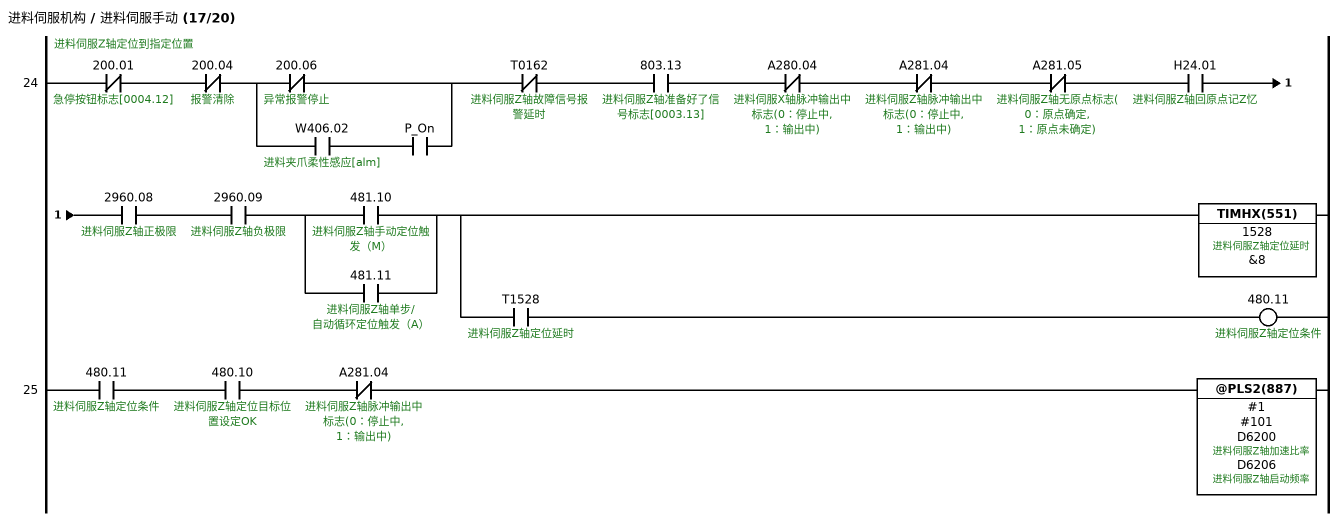
; [picture p96: 进料伺服机构 / 进料伺服手动, rungs 24-25]
; rung 24: 进料伺服Z轴定位到指定位置
LDNOT 200.01  ; 急停按钮标志[0004.12]
ANDNOT 200.04  ; 报警清除
LDNOT 200.06  ; 异常报警停止
LD W406.02  ; 进料夹爪柔性感应[alm]
AND P_On
ORLD
ANDLD
ANDNOT T0162  ; 进料伺服Z轴故障信号报警延时
AND 803.13  ; 进料伺服Z轴准备好了信号标志[0003.13]
ANDNOT A280.04  ; 进料伺服X轴脉冲输出中标志(0：停止中,1：输出中)
ANDNOT A281.04  ; 进料伺服Z轴脉冲输出中标志(0：停止中,1：输出中)
ANDNOT A281.05  ; 进料伺服Z轴无原点标志(0：原点确定,1：原点未确定)
AND H24.01  ; 进料伺服Z轴回原点记Z忆
AND 2960.08  ; 进料伺服Z轴正极限
AND 2960.09  ; 进料伺服Z轴负极限
LD 481.10  ; 进料伺服Z轴手动定位触发（M）
OR 481.11  ; 进料伺服Z轴单步/自动循环定位触发（A）
ANDLD
TIMHX(551) 1528 &8  ; 进料伺服Z轴定位延时
AND T1528  ; 进料伺服Z轴定位延时
OUT 480.11  ; 进料伺服Z轴定位条件
; rung 25
LD 480.11  ; 进料伺服Z轴定位条件
AND 480.10  ; 进料伺服Z轴定位目标位置设定OK
ANDNOT A281.04  ; 进料伺服Z轴脉冲输出中标志(0：停止中,1：输出中)
@PLS2(887) #1 #101 D6200 D6206  ; 进料伺服Z轴加速比率, 进料伺服Z轴启动频率

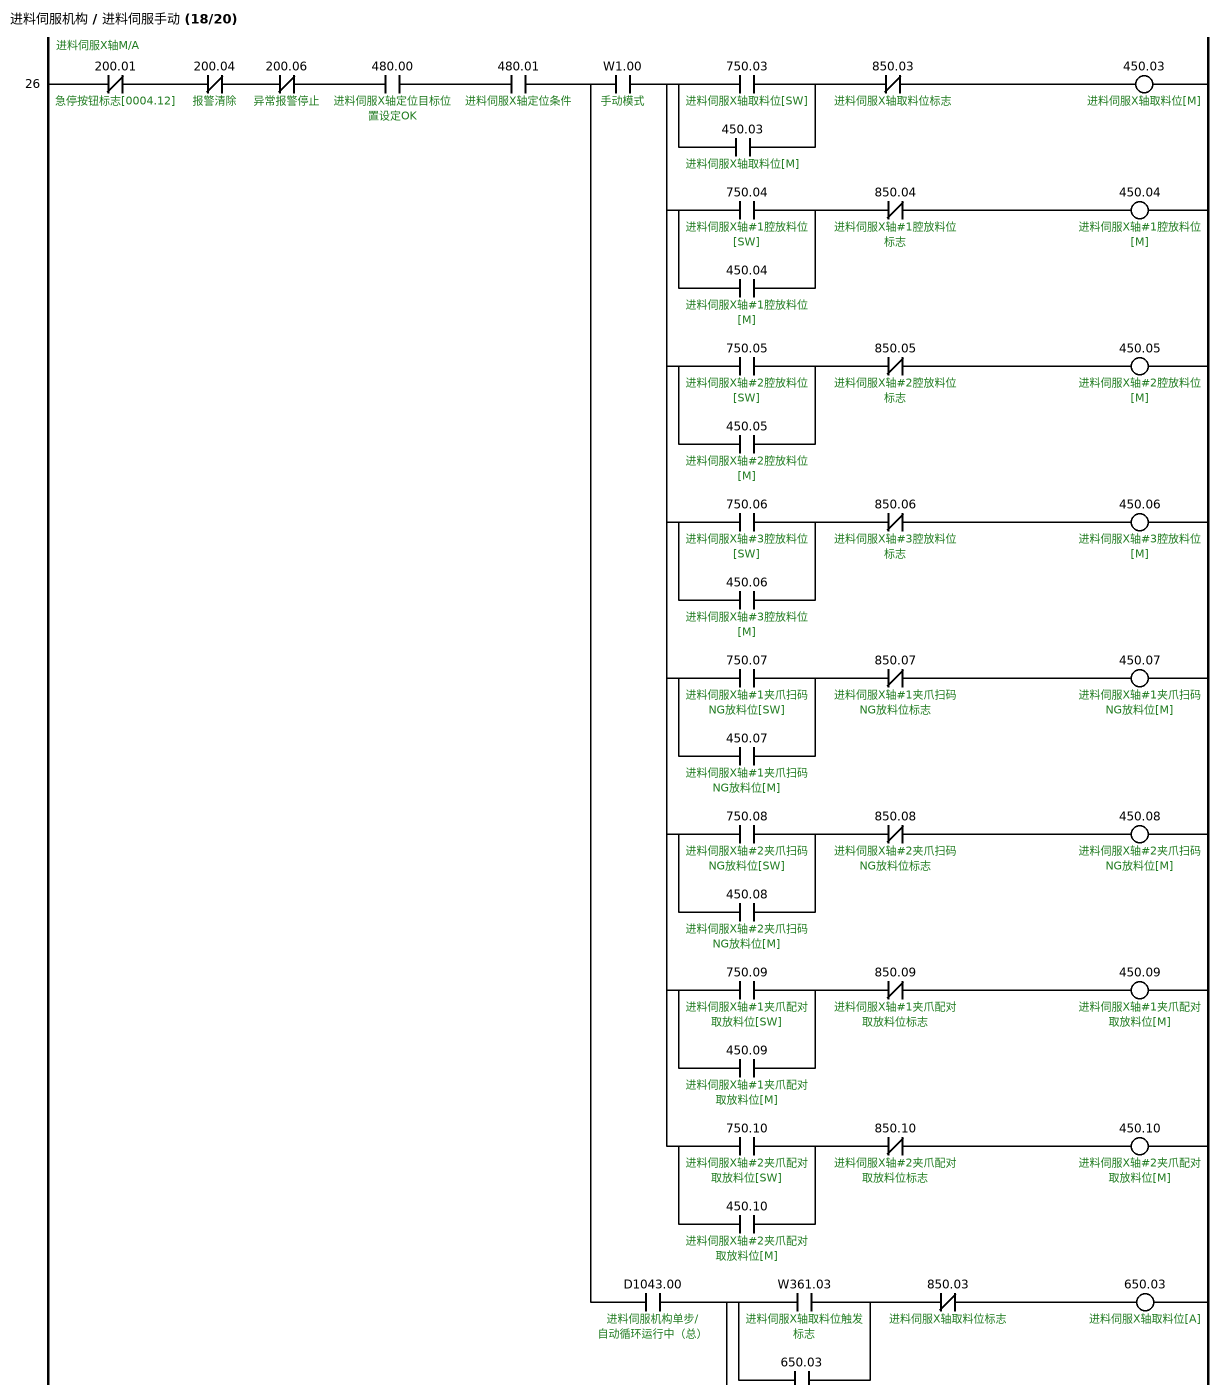

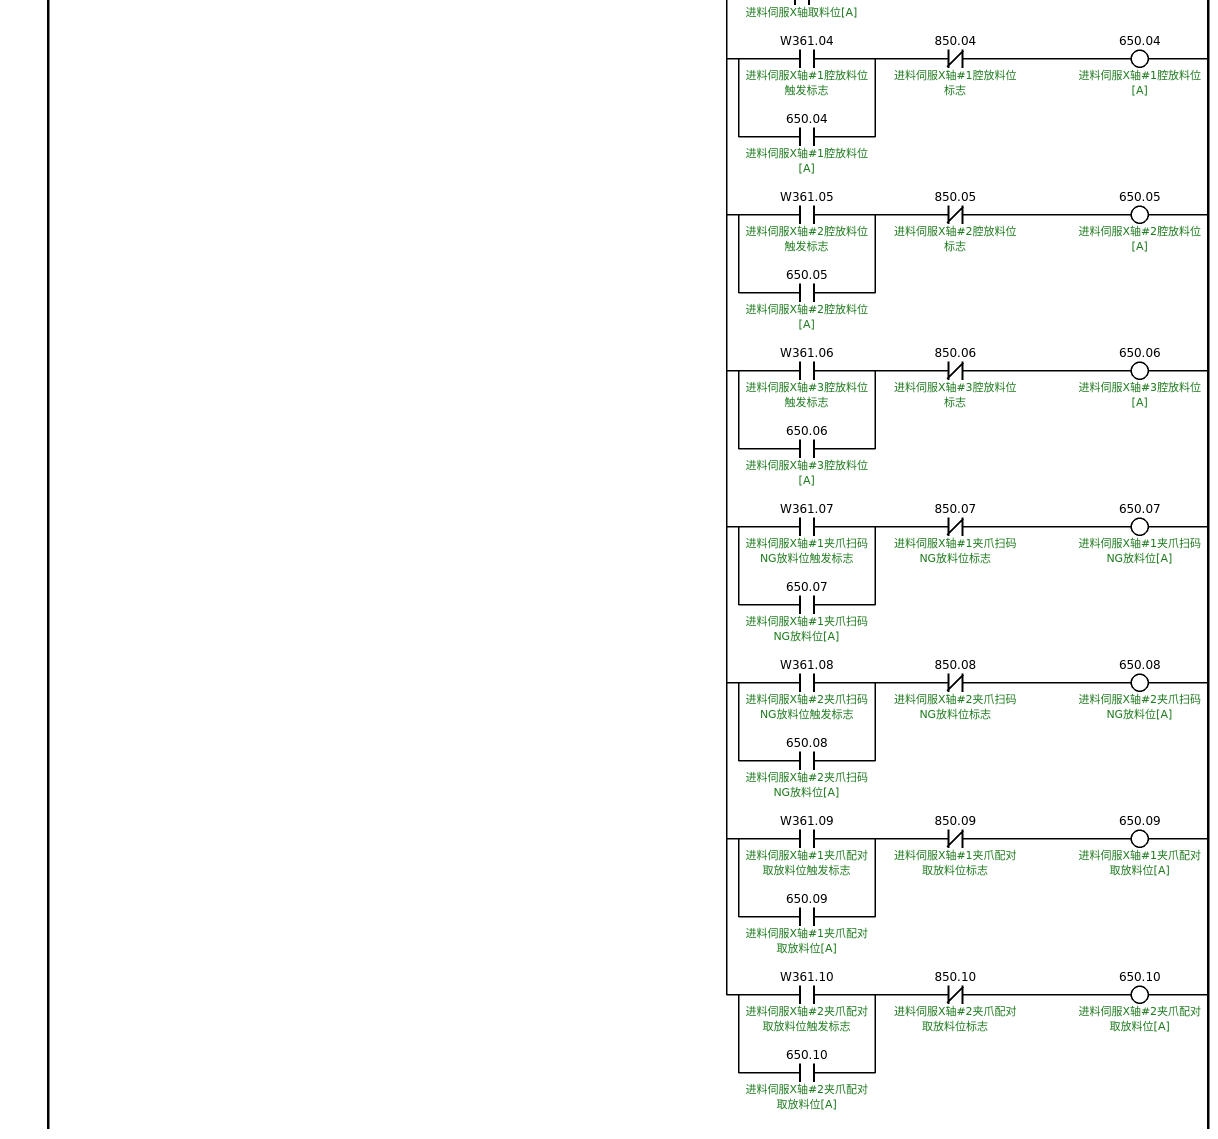
; rung 26: 进料伺服X轴M/A
LDNOT 200.01  ; 急停按钮标志[0004.12]
ANDNOT 200.04  ; 报警清除
ANDNOT 200.06  ; 异常报警停止
AND 480.00  ; 进料伺服X轴定位目标位置设定OK
AND 480.01  ; 进料伺服X轴定位条件
OUT TR0
AND W1.00  ; 手动模式
OUT TR1
LD 750.03  ; 进料伺服X轴取料位[SW]
OR 450.03  ; 进料伺服X轴取料位[M]
ANDLD
ANDNOT 850.03  ; 进料伺服X轴取料位标志
OUT 450.03  ; 进料伺服X轴取料位[M]
LD TR1
LD 750.04  ; 进料伺服X轴#1腔放料位[SW]
OR 450.04  ; 进料伺服X轴#1腔放料位[M]
ANDLD
ANDNOT 850.04  ; 进料伺服X轴#1腔放料位标志
OUT 450.04  ; 进料伺服X轴#1腔放料位[M]
LD TR1
LD 750.05  ; 进料伺服X轴#2腔放料位[SW]
OR 450.05  ; 进料伺服X轴#2腔放料位[M]
ANDLD
ANDNOT 850.05  ; 进料伺服X轴#2腔放料位标志
OUT 450.05  ; 进料伺服X轴#2腔放料位[M]
LD TR1
LD 750.06  ; 进料伺服X轴#3腔放料位[SW]
OR 450.06  ; 进料伺服X轴#3腔放料位[M]
ANDLD
ANDNOT 850.06  ; 进料伺服X轴#3腔放料位标志
OUT 450.06  ; 进料伺服X轴#3腔放料位[M]
LD TR1
LD 750.07  ; 进料伺服X轴#1夹爪扫码NG放料位[SW]
OR 450.07  ; 进料伺服X轴#1夹爪扫码NG放料位[M]
ANDLD
ANDNOT 850.07  ; 进料伺服X轴#1夹爪扫码NG放料位标志
OUT 450.07  ; 进料伺服X轴#1夹爪扫码NG放料位[M]
LD TR1
LD 750.08  ; 进料伺服X轴#2夹爪扫码NG放料位[SW]
OR 450.08  ; 进料伺服X轴#2夹爪扫码NG放料位[M]
ANDLD
ANDNOT 850.08  ; 进料伺服X轴#2夹爪扫码NG放料位标志
OUT 450.08  ; 进料伺服X轴#2夹爪扫码NG放料位[M]
LD TR1
LD 750.09  ; 进料伺服X轴#1夹爪配对取放料位[SW]
OR 450.09  ; 进料伺服X轴#1夹爪配对取放料位[M]
ANDLD
ANDNOT 850.09  ; 进料伺服X轴#1夹爪配对取放料位标志
OUT 450.09  ; 进料伺服X轴#1夹爪配对取放料位[M]
LD TR1
LD 750.10  ; 进料伺服X轴#2夹爪配对取放料位[SW]
OR 450.10  ; 进料伺服X轴#2夹爪配对取放料位[M]
ANDLD
ANDNOT 850.10  ; 进料伺服X轴#2夹爪配对取放料位标志
OUT 450.10  ; 进料伺服X轴#2夹爪配对取放料位[M]
LD TR0
AND D1043.00  ; 进料伺服机构单步/自动循环运行中（总）
OUT TR0
LD W361.03  ; 进料伺服X轴取料位触发标志
OR 650.03  ; 进料伺服X轴取料位[A]
ANDLD
ANDNOT 850.03  ; 进料伺服X轴取料位标志
OUT 650.03  ; 进料伺服X轴取料位[A]
LD TR0
LD W361.04  ; 进料伺服X轴#1腔放料位触发标志
OR 650.04  ; 进料伺服X轴#1腔放料位[A]
ANDLD
ANDNOT 850.04  ; 进料伺服X轴#1腔放料位标志
OUT 650.04  ; 进料伺服X轴#1腔放料位[A]
LD TR0
LD W361.05  ; 进料伺服X轴#2腔放料位触发标志
OR 650.05  ; 进料伺服X轴#2腔放料位[A]
ANDLD
ANDNOT 850.05  ; 进料伺服X轴#2腔放料位标志
OUT 650.05  ; 进料伺服X轴#2腔放料位[A]
LD TR0
LD W361.06  ; 进料伺服X轴#3腔放料位触发标志
OR 650.06  ; 进料伺服X轴#3腔放料位[A]
ANDLD
ANDNOT 850.06  ; 进料伺服X轴#3腔放料位标志
OUT 650.06  ; 进料伺服X轴#3腔放料位[A]
LD TR0
LD W361.07  ; 进料伺服X轴#1夹爪扫码NG放料位触发标志
OR 650.07  ; 进料伺服X轴#1夹爪扫码NG放料位[A]
ANDLD
ANDNOT 850.07  ; 进料伺服X轴#1夹爪扫码NG放料位标志
OUT 650.07  ; 进料伺服X轴#1夹爪扫码NG放料位[A]
LD TR0
LD W361.08  ; 进料伺服X轴#2夹爪扫码NG放料位触发标志
OR 650.08  ; 进料伺服X轴#2夹爪扫码NG放料位[A]
ANDLD
ANDNOT 850.08  ; 进料伺服X轴#2夹爪扫码NG放料位标志
OUT 650.08  ; 进料伺服X轴#2夹爪扫码NG放料位[A]
LD TR0
LD W361.09  ; 进料伺服X轴#1夹爪配对取放料位触发标志
OR 650.09  ; 进料伺服X轴#1夹爪配对取放料位[A]
ANDLD
ANDNOT 850.09  ; 进料伺服X轴#1夹爪配对取放料位标志
OUT 650.09  ; 进料伺服X轴#1夹爪配对取放料位[A]
LD TR0
LD W361.10  ; 进料伺服X轴#2夹爪配对取放料位触发标志
OR 650.10  ; 进料伺服X轴#2夹爪配对取放料位[A]
ANDLD
ANDNOT 850.10  ; 进料伺服X轴#2夹爪配对取放料位标志
OUT 650.10  ; 进料伺服X轴#2夹爪配对取放料位[A]

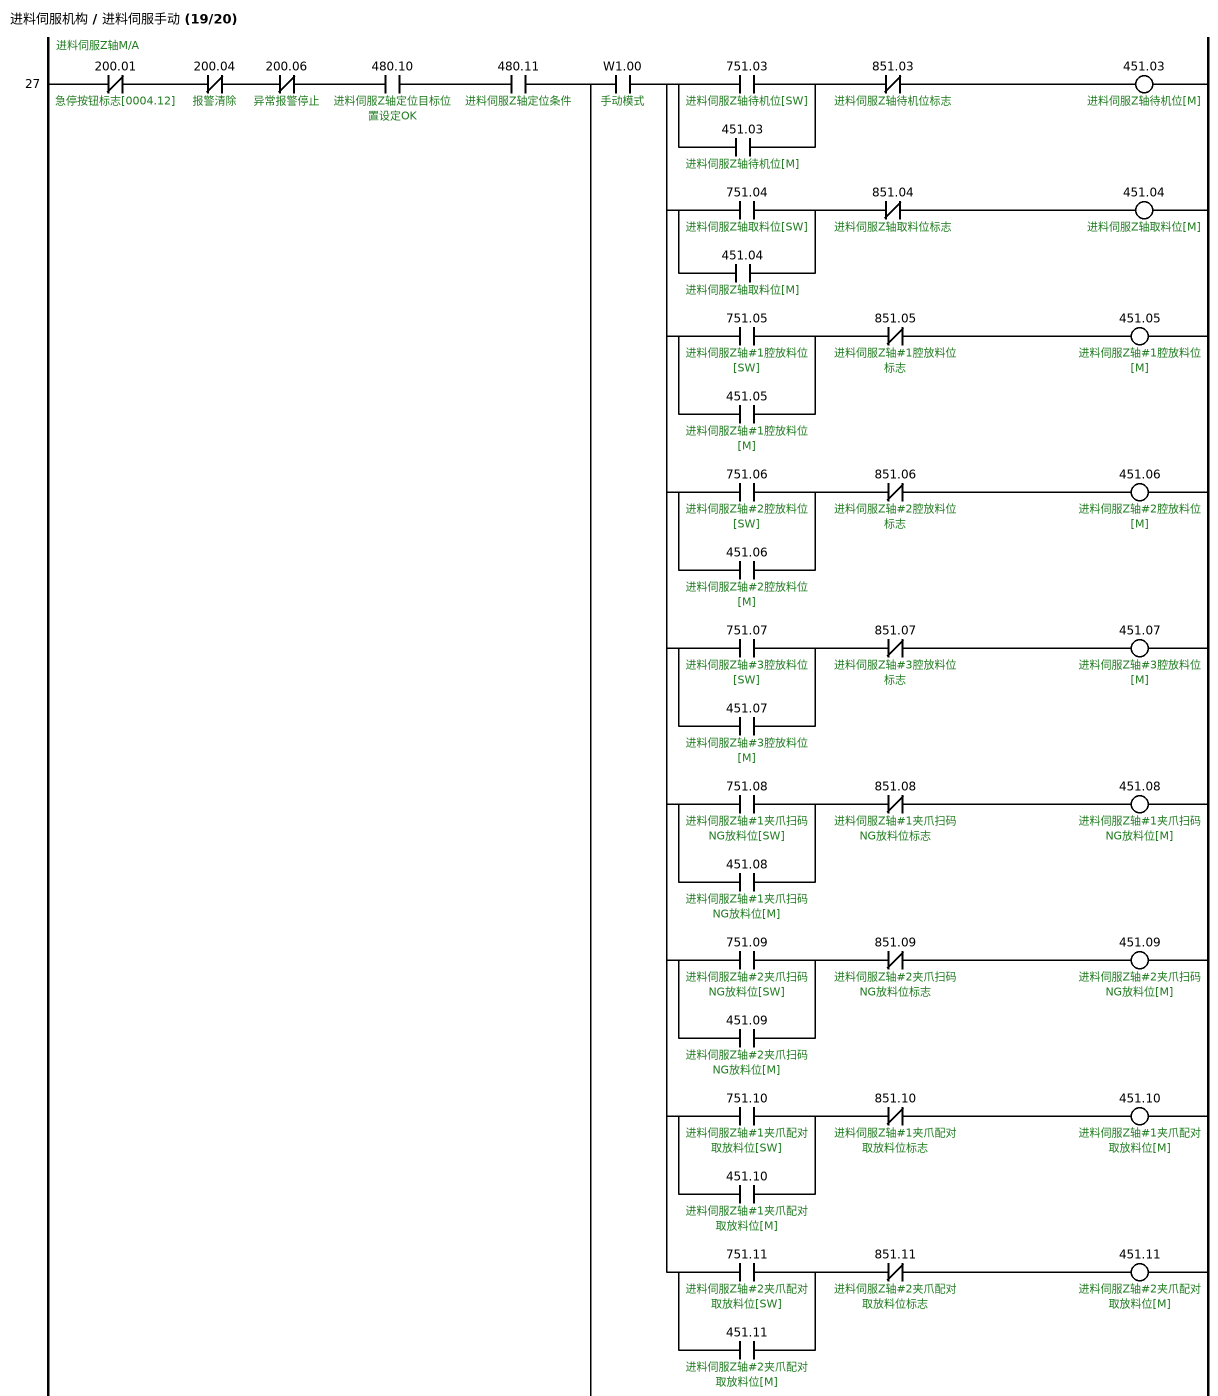

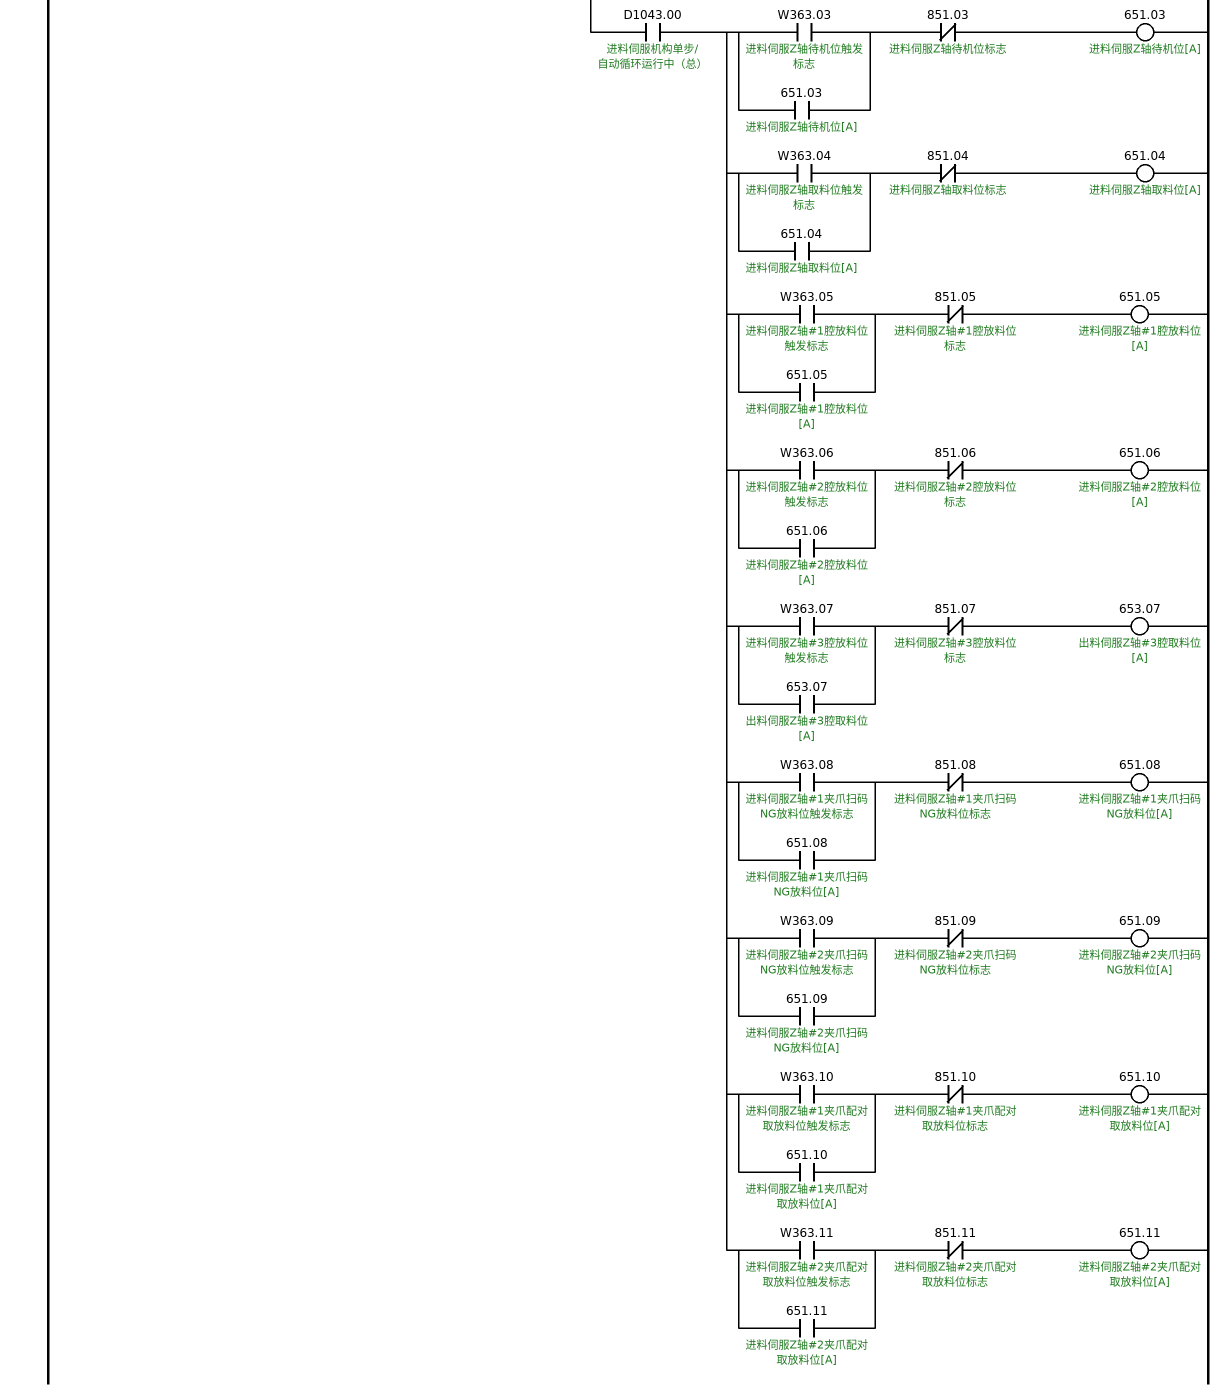
; rung 27: 进料伺服Z轴M/A
LDNOT 200.01  ; 急停按钮标志[0004.12]
ANDNOT 200.04  ; 报警清除
ANDNOT 200.06  ; 异常报警停止
AND 480.10  ; 进料伺服Z轴定位目标位置设定OK
AND 480.11  ; 进料伺服Z轴定位条件
OUT TR0
AND W1.00  ; 手动模式
OUT TR1
LD 751.03  ; 进料伺服Z轴待机位[SW]
OR 451.03  ; 进料伺服Z轴待机位[M]
ANDLD
ANDNOT 851.03  ; 进料伺服Z轴待机位标志
OUT 451.03  ; 进料伺服Z轴待机位[M]
LD TR1
LD 751.04  ; 进料伺服Z轴取料位[SW]
OR 451.04  ; 进料伺服Z轴取料位[M]
ANDLD
ANDNOT 851.04  ; 进料伺服Z轴取料位标志
OUT 451.04  ; 进料伺服Z轴取料位[M]
LD TR1
LD 751.05  ; 进料伺服Z轴#1腔放料位[SW]
OR 451.05  ; 进料伺服Z轴#1腔放料位[M]
ANDLD
ANDNOT 851.05  ; 进料伺服Z轴#1腔放料位标志
OUT 451.05  ; 进料伺服Z轴#1腔放料位[M]
LD TR1
LD 751.06  ; 进料伺服Z轴#2腔放料位[SW]
OR 451.06  ; 进料伺服Z轴#2腔放料位[M]
ANDLD
ANDNOT 851.06  ; 进料伺服Z轴#2腔放料位标志
OUT 451.06  ; 进料伺服Z轴#2腔放料位[M]
LD TR1
LD 751.07  ; 进料伺服Z轴#3腔放料位[SW]
OR 451.07  ; 进料伺服Z轴#3腔放料位[M]
ANDLD
ANDNOT 851.07  ; 进料伺服Z轴#3腔放料位标志
OUT 451.07  ; 进料伺服Z轴#3腔放料位[M]
LD TR1
LD 751.08  ; 进料伺服Z轴#1夹爪扫码NG放料位[SW]
OR 451.08  ; 进料伺服Z轴#1夹爪扫码NG放料位[M]
ANDLD
ANDNOT 851.08  ; 进料伺服Z轴#1夹爪扫码NG放料位标志
OUT 451.08  ; 进料伺服Z轴#1夹爪扫码NG放料位[M]
LD TR1
LD 751.09  ; 进料伺服Z轴#2夹爪扫码NG放料位[SW]
OR 451.09  ; 进料伺服Z轴#2夹爪扫码NG放料位[M]
ANDLD
ANDNOT 851.09  ; 进料伺服Z轴#2夹爪扫码NG放料位标志
OUT 451.09  ; 进料伺服Z轴#2夹爪扫码NG放料位[M]
LD TR1
LD 751.10  ; 进料伺服Z轴#1夹爪配对取放料位[SW]
OR 451.10  ; 进料伺服Z轴#1夹爪配对取放料位[M]
ANDLD
ANDNOT 851.10  ; 进料伺服Z轴#1夹爪配对取放料位标志
OUT 451.10  ; 进料伺服Z轴#1夹爪配对取放料位[M]
LD TR1
LD 751.11  ; 进料伺服Z轴#2夹爪配对取放料位[SW]
OR 451.11  ; 进料伺服Z轴#2夹爪配对取放料位[M]
ANDLD
ANDNOT 851.11  ; 进料伺服Z轴#2夹爪配对取放料位标志
OUT 451.11  ; 进料伺服Z轴#2夹爪配对取放料位[M]
LD TR0
AND D1043.00  ; 进料伺服机构单步/自动循环运行中（总）
OUT TR0
LD W363.03  ; 进料伺服Z轴待机位触发标志
OR 651.03  ; 进料伺服Z轴待机位[A]
ANDLD
ANDNOT 851.03  ; 进料伺服Z轴待机位标志
OUT 651.03  ; 进料伺服Z轴待机位[A]
LD TR0
LD W363.04  ; 进料伺服Z轴取料位触发标志
OR 651.04  ; 进料伺服Z轴取料位[A]
ANDLD
ANDNOT 851.04  ; 进料伺服Z轴取料位标志
OUT 651.04  ; 进料伺服Z轴取料位[A]
LD TR0
LD W363.05  ; 进料伺服Z轴#1腔放料位触发标志
OR 651.05  ; 进料伺服Z轴#1腔放料位[A]
ANDLD
ANDNOT 851.05  ; 进料伺服Z轴#1腔放料位标志
OUT 651.05  ; 进料伺服Z轴#1腔放料位[A]
LD TR0
LD W363.06  ; 进料伺服Z轴#2腔放料位触发标志
OR 651.06  ; 进料伺服Z轴#2腔放料位[A]
ANDLD
ANDNOT 851.06  ; 进料伺服Z轴#2腔放料位标志
OUT 651.06  ; 进料伺服Z轴#2腔放料位[A]
LD TR0
LD W363.07  ; 进料伺服Z轴#3腔放料位触发标志
OR 653.07  ; 出料伺服Z轴#3腔取料位[A]
ANDLD
ANDNOT 851.07  ; 进料伺服Z轴#3腔放料位标志
OUT 653.07  ; 出料伺服Z轴#3腔取料位[A]
LD TR0
LD W363.08  ; 进料伺服Z轴#1夹爪扫码NG放料位触发标志
OR 651.08  ; 进料伺服Z轴#1夹爪扫码NG放料位[A]
ANDLD
ANDNOT 851.08  ; 进料伺服Z轴#1夹爪扫码NG放料位标志
OUT 651.08  ; 进料伺服Z轴#1夹爪扫码NG放料位[A]
LD TR0
LD W363.09  ; 进料伺服Z轴#2夹爪扫码NG放料位触发标志
OR 651.09  ; 进料伺服Z轴#2夹爪扫码NG放料位[A]
ANDLD
ANDNOT 851.09  ; 进料伺服Z轴#2夹爪扫码NG放料位标志
OUT 651.09  ; 进料伺服Z轴#2夹爪扫码NG放料位[A]
LD TR0
LD W363.10  ; 进料伺服Z轴#1夹爪配对取放料位触发标志
OR 651.10  ; 进料伺服Z轴#1夹爪配对取放料位[A]
ANDLD
ANDNOT 851.10  ; 进料伺服Z轴#1夹爪配对取放料位标志
OUT 651.10  ; 进料伺服Z轴#1夹爪配对取放料位[A]
LD TR0
LD W363.11  ; 进料伺服Z轴#2夹爪配对取放料位触发标志
OR 651.11  ; 进料伺服Z轴#2夹爪配对取放料位[A]
ANDLD
ANDNOT 851.11  ; 进料伺服Z轴#2夹爪配对取放料位标志
OUT 651.11  ; 进料伺服Z轴#2夹爪配对取放料位[A]

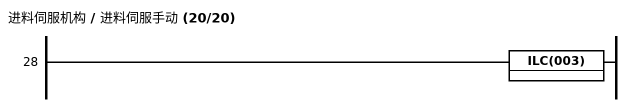
; rung 28
ILC(003)

### Section 进料伺服自动

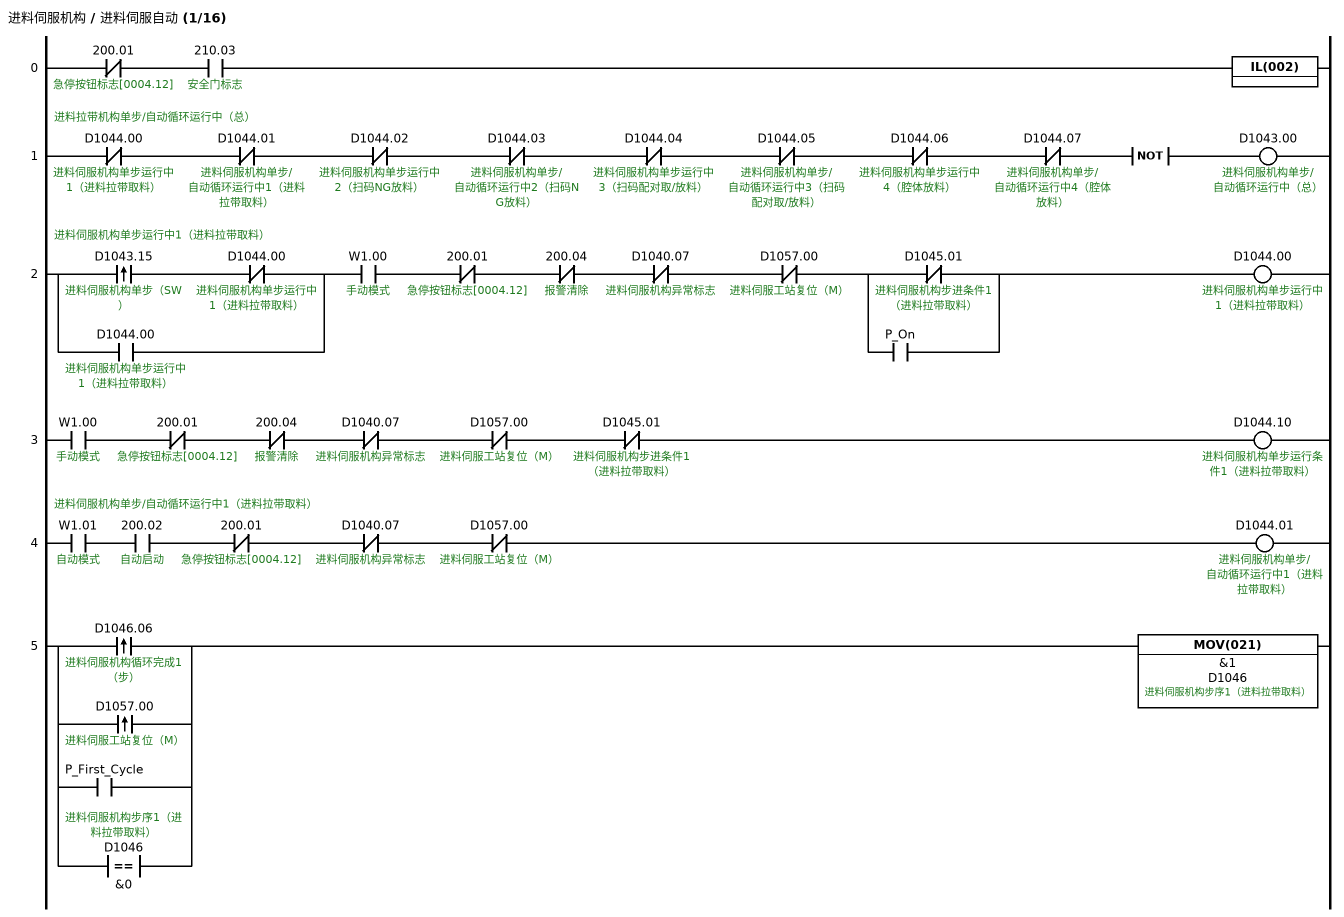
; rung 0
LDNOT 200.01  ; 急停按钮标志[0004.12]
AND 210.03  ; 安全门标志
IL(002)
; rung 1: 进料拉带机构单步/自动循环运行中（总）
LDNOT D1044.00  ; 进料伺服机构单步运行中1（进料拉带取料）
ANDNOT D1044.01  ; 进料伺服机构单步/自动循环运行中1（进料拉带取料）
ANDNOT D1044.02  ; 进料伺服机构单步运行中2（扫码NG放料）
ANDNOT D1044.03  ; 进料伺服机构单步/自动循环运行中2（扫码NG放料）
ANDNOT D1044.04  ; 进料伺服机构单步运行中3（扫码配对取/放料）
ANDNOT D1044.05  ; 进料伺服机构单步/自动循环运行中3（扫码配对取/放料）
ANDNOT D1044.06  ; 进料伺服机构单步运行中4（腔体放料）
ANDNOT D1044.07  ; 进料伺服机构单步/自动循环运行中4（腔体放料）
NOT(520)
OUT D1043.00  ; 进料伺服机构单步/自动循环运行中（总）
; rung 2: 进料伺服机构单步运行中1（进料拉带取料）
@LD D1043.15  ; 进料伺服机构单步（SW）
ANDNOT D1044.00  ; 进料伺服机构单步运行中1（进料拉带取料）
OR D1044.00  ; 进料伺服机构单步运行中1（进料拉带取料）
AND W1.00  ; 手动模式
ANDNOT 200.01  ; 急停按钮标志[0004.12]
ANDNOT 200.04  ; 报警清除
ANDNOT D1040.07  ; 进料伺服机构异常标志
ANDNOT D1057.00  ; 进料伺服工站复位（M）
LDNOT D1045.01  ; 进料伺服机构步进条件1（进料拉带取料）
OR P_On
ANDLD
OUT D1044.00  ; 进料伺服机构单步运行中1（进料拉带取料）
; rung 3
LD W1.00  ; 手动模式
ANDNOT 200.01  ; 急停按钮标志[0004.12]
ANDNOT 200.04  ; 报警清除
ANDNOT D1040.07  ; 进料伺服机构异常标志
ANDNOT D1057.00  ; 进料伺服工站复位（M）
ANDNOT D1045.01  ; 进料伺服机构步进条件1（进料拉带取料）
OUT D1044.10  ; 进料伺服机构单步运行条件1（进料拉带取料）
; rung 4: 进料伺服机构单步/自动循环运行中1（进料拉带取料）
LD W1.01  ; 自动模式
AND 200.02  ; 自动启动
ANDNOT 200.01  ; 急停按钮标志[0004.12]
ANDNOT D1040.07  ; 进料伺服机构异常标志
ANDNOT D1057.00  ; 进料伺服工站复位（M）
OUT D1044.01  ; 进料伺服机构单步/自动循环运行中1（进料拉带取料）
; rung 5
@LD D1046.06  ; 进料伺服机构循环完成1（步）
@OR D1057.00  ; 进料伺服工站复位（M）
OR P_First_Cycle
OR=(300) D1046 &0  ; 进料伺服机构步序1（进料拉带取料）
MOV(021) &1 D1046  ; 进料伺服机构步序1（进料拉带取料）

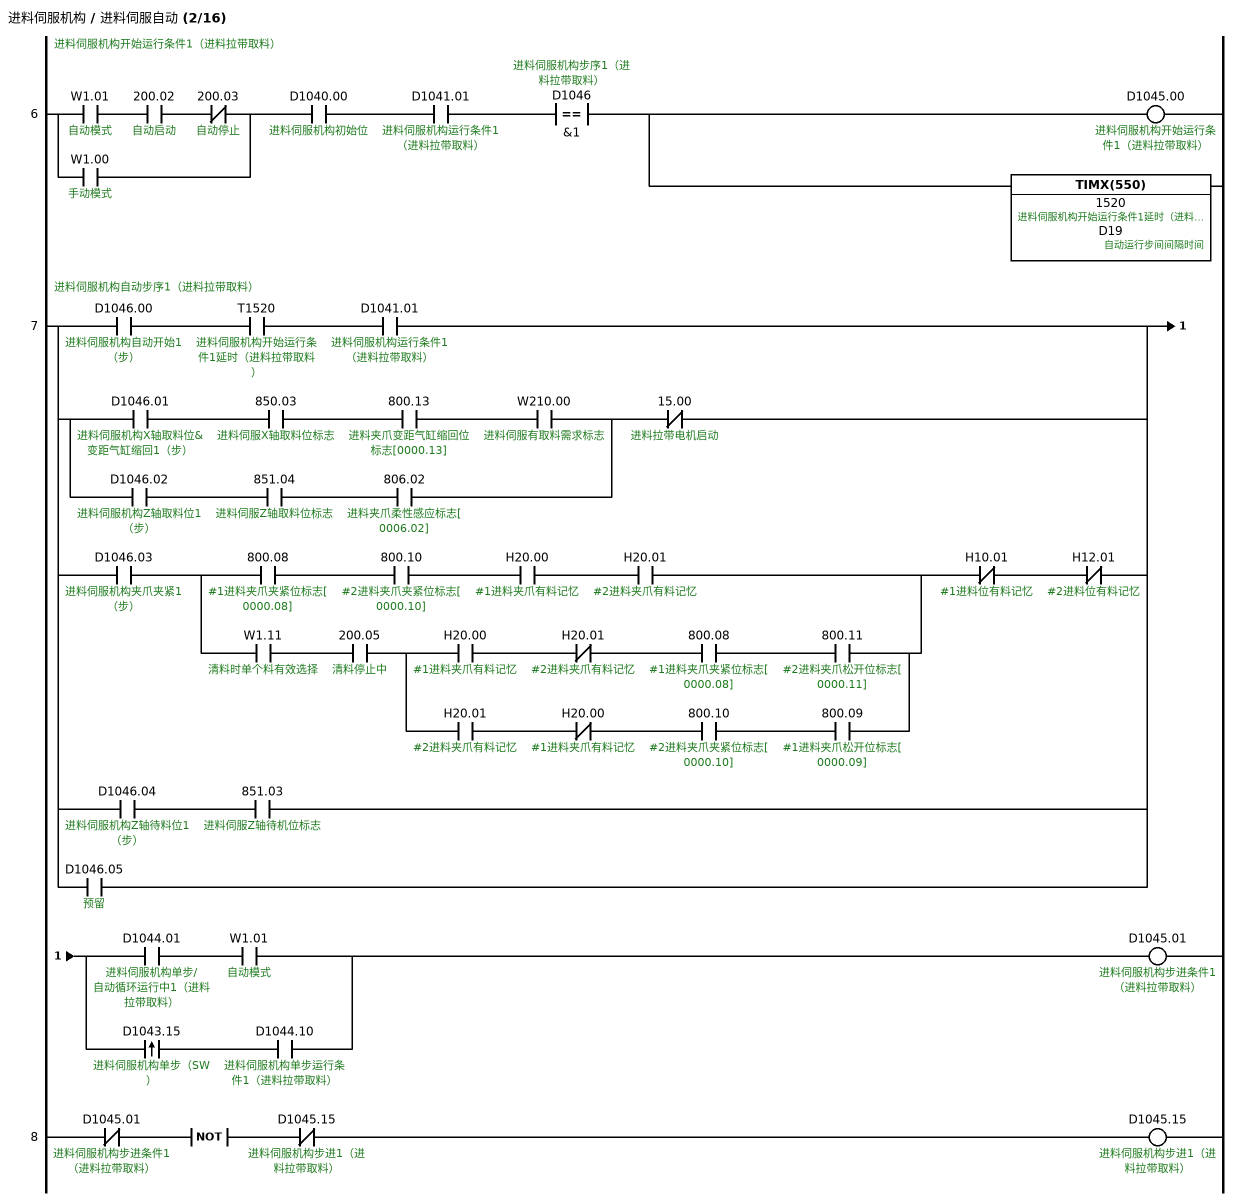
; rung 6: 进料伺服机构开始运行条件1（进料拉带取料）
LD W1.01  ; 自动模式
AND 200.02  ; 自动启动
ANDNOT 200.03  ; 自动停止
OR W1.00  ; 手动模式
AND D1040.00  ; 进料伺服机构初始位
AND D1041.01  ; 进料伺服机构运行条件1（进料拉带取料）
AND=(300) D1046 &1  ; 进料伺服机构步序1（进料拉带取料）
OUT D1045.00  ; 进料伺服机构开始运行条件1（进料拉带取料）
TIMX(550) 1520 D19  ; 自动运行步间间隔时间, 进料伺服机构开始运行条件1延时（进料拉带取料）
; rung 7: 进料伺服机构自动步序1（进料拉带取料）
LD D1046.00  ; 进料伺服机构自动开始1（步）
AND T1520  ; 进料伺服机构开始运行条件1延时（进料拉带取料）
AND D1041.01  ; 进料伺服机构运行条件1（进料拉带取料）
LD D1046.01  ; 进料伺服机构X轴取料位&变距气缸缩回1（步）
AND 850.03  ; 进料伺服X轴取料位标志
AND 800.13  ; 进料夹爪变距气缸缩回位标志[0000.13]
AND W210.00  ; 进料伺服有取料需求标志
LD D1046.02  ; 进料伺服机构Z轴取料位1（步）
AND 851.04  ; 进料伺服Z轴取料位标志
AND 806.02  ; 进料夹爪柔性感应标志[0006.02]
ORLD
ANDNOT 15.00  ; 进料拉带电机启动
ORLD
LD D1046.03  ; 进料伺服机构夹爪夹紧1（步）
LD 800.08  ; #1进料夹爪夹紧位标志[0000.08]
AND 800.10  ; #2进料夹爪夹紧位标志[0000.10]
AND H20.00  ; #1进料夹爪有料记忆
AND H20.01  ; #2进料夹爪有料记忆
LD W1.11  ; 清料时单个料有效选择
AND 200.05  ; 清料停止中
LD H20.00  ; #1进料夹爪有料记忆
ANDNOT H20.01  ; #2进料夹爪有料记忆
AND 800.08  ; #1进料夹爪夹紧位标志[0000.08]
AND 800.11  ; #2进料夹爪松开位标志[0000.11]
LD H20.01  ; #2进料夹爪有料记忆
ANDNOT H20.00  ; #1进料夹爪有料记忆
AND 800.10  ; #2进料夹爪夹紧位标志[0000.10]
AND 800.09  ; #1进料夹爪松开位标志[0000.09]
ORLD
ANDLD
ORLD
ANDLD
ANDNOT H10.01  ; #1进料位有料记忆
ANDNOT H12.01  ; #2进料位有料记忆
ORLD
LD D1046.04  ; 进料伺服机构Z轴待料位1（步）
AND 851.03  ; 进料伺服Z轴待机位标志
ORLD
OR D1046.05  ; 预留
LD D1044.01  ; 进料伺服机构单步/自动循环运行中1（进料拉带取料）
AND W1.01  ; 自动模式
@LD D1043.15  ; 进料伺服机构单步（SW）
AND D1044.10  ; 进料伺服机构单步运行条件1（进料拉带取料）
ORLD
ANDLD
OUT D1045.01  ; 进料伺服机构步进条件1（进料拉带取料）
; rung 8
LDNOT D1045.01  ; 进料伺服机构步进条件1（进料拉带取料）
NOT(520)
ANDNOT D1045.15  ; 进料伺服机构步进1（进料拉带取料）
OUT D1045.15  ; 进料伺服机构步进1（进料拉带取料）

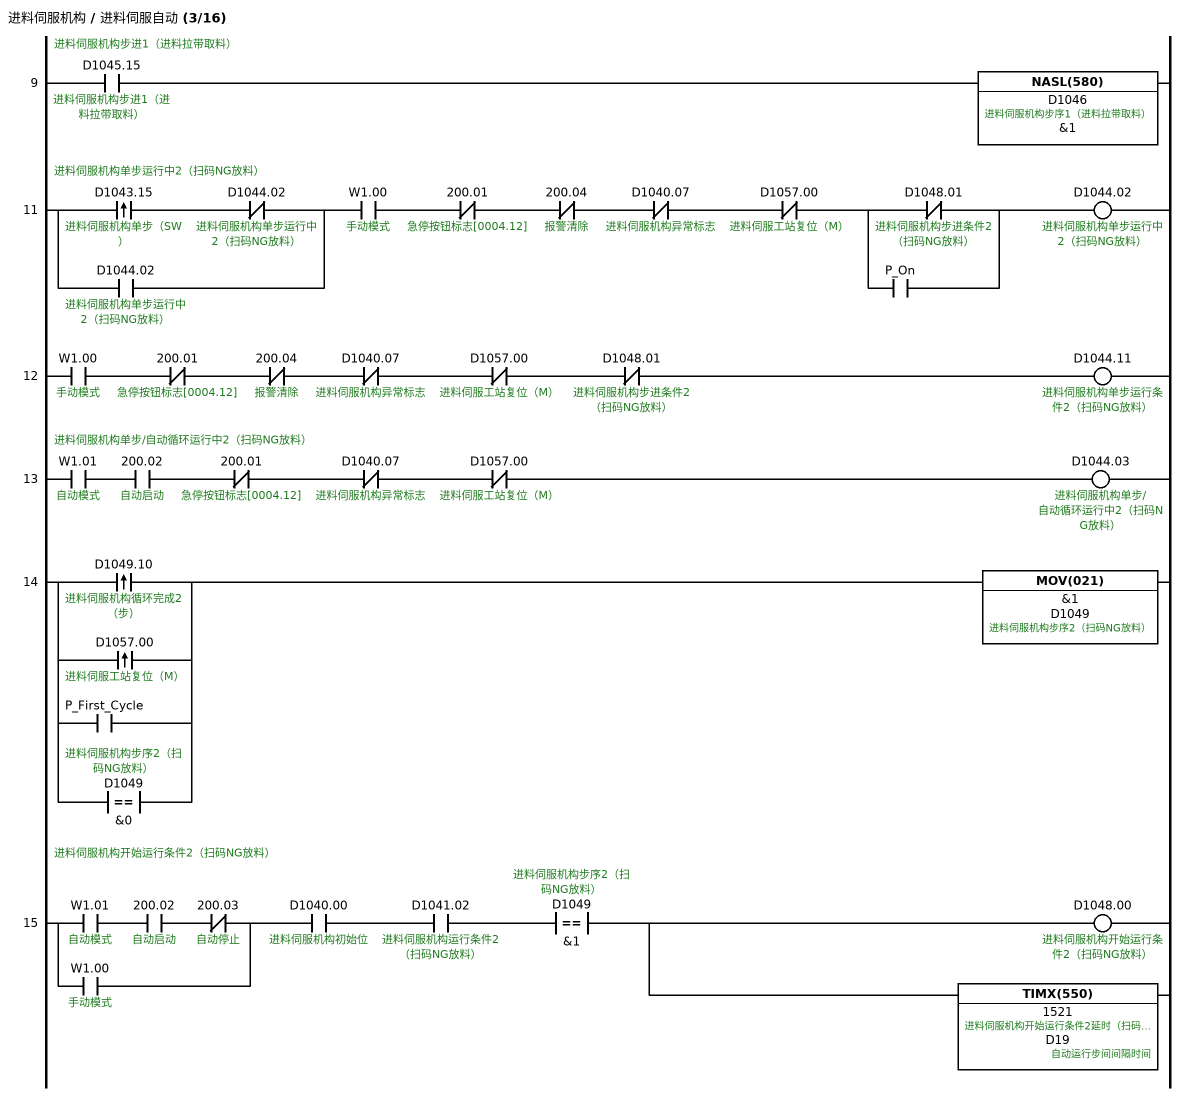
; rung 9: 进料伺服机构步进1（进料拉带取料）
LD D1045.15  ; 进料伺服机构步进1（进料拉带取料）
NASL(580) D1046 &1  ; 进料伺服机构步序1（进料拉带取料）
; rung 10: 进料伺服机构步序跳转程序1（进料拉带取料）
; rung 11: 进料伺服机构单步运行中2（扫码NG放料）
@LD D1043.15  ; 进料伺服机构单步（SW）
ANDNOT D1044.02  ; 进料伺服机构单步运行中2（扫码NG放料）
OR D1044.02  ; 进料伺服机构单步运行中2（扫码NG放料）
AND W1.00  ; 手动模式
ANDNOT 200.01  ; 急停按钮标志[0004.12]
ANDNOT 200.04  ; 报警清除
ANDNOT D1040.07  ; 进料伺服机构异常标志
ANDNOT D1057.00  ; 进料伺服工站复位（M）
LDNOT D1048.01  ; 进料伺服机构步进条件2（扫码NG放料）
OR P_On
ANDLD
OUT D1044.02  ; 进料伺服机构单步运行中2（扫码NG放料）
; rung 12
LD W1.00  ; 手动模式
ANDNOT 200.01  ; 急停按钮标志[0004.12]
ANDNOT 200.04  ; 报警清除
ANDNOT D1040.07  ; 进料伺服机构异常标志
ANDNOT D1057.00  ; 进料伺服工站复位（M）
ANDNOT D1048.01  ; 进料伺服机构步进条件2（扫码NG放料）
OUT D1044.11  ; 进料伺服机构单步运行条件2（扫码NG放料）
; rung 13: 进料伺服机构单步/自动循环运行中2（扫码NG放料）
LD W1.01  ; 自动模式
AND 200.02  ; 自动启动
ANDNOT 200.01  ; 急停按钮标志[0004.12]
ANDNOT D1040.07  ; 进料伺服机构异常标志
ANDNOT D1057.00  ; 进料伺服工站复位（M）
OUT D1044.03  ; 进料伺服机构单步/自动循环运行中2（扫码NG放料）
; rung 14
@LD D1049.10  ; 进料伺服机构循环完成2（步）
@OR D1057.00  ; 进料伺服工站复位（M）
OR P_First_Cycle
OR=(300) D1049 &0  ; 进料伺服机构步序2（扫码NG放料）
MOV(021) &1 D1049  ; 进料伺服机构步序2（扫码NG放料）
; rung 15: 进料伺服机构开始运行条件2（扫码NG放料）
LD W1.01  ; 自动模式
AND 200.02  ; 自动启动
ANDNOT 200.03  ; 自动停止
OR W1.00  ; 手动模式
AND D1040.00  ; 进料伺服机构初始位
AND D1041.02  ; 进料伺服机构运行条件2（扫码NG放料）
AND=(300) D1049 &1  ; 进料伺服机构步序2（扫码NG放料）
OUT D1048.00  ; 进料伺服机构开始运行条件2（扫码NG放料）
TIMX(550) 1521 D19  ; 自动运行步间间隔时间, 进料伺服机构开始运行条件2延时（扫码NG放料）

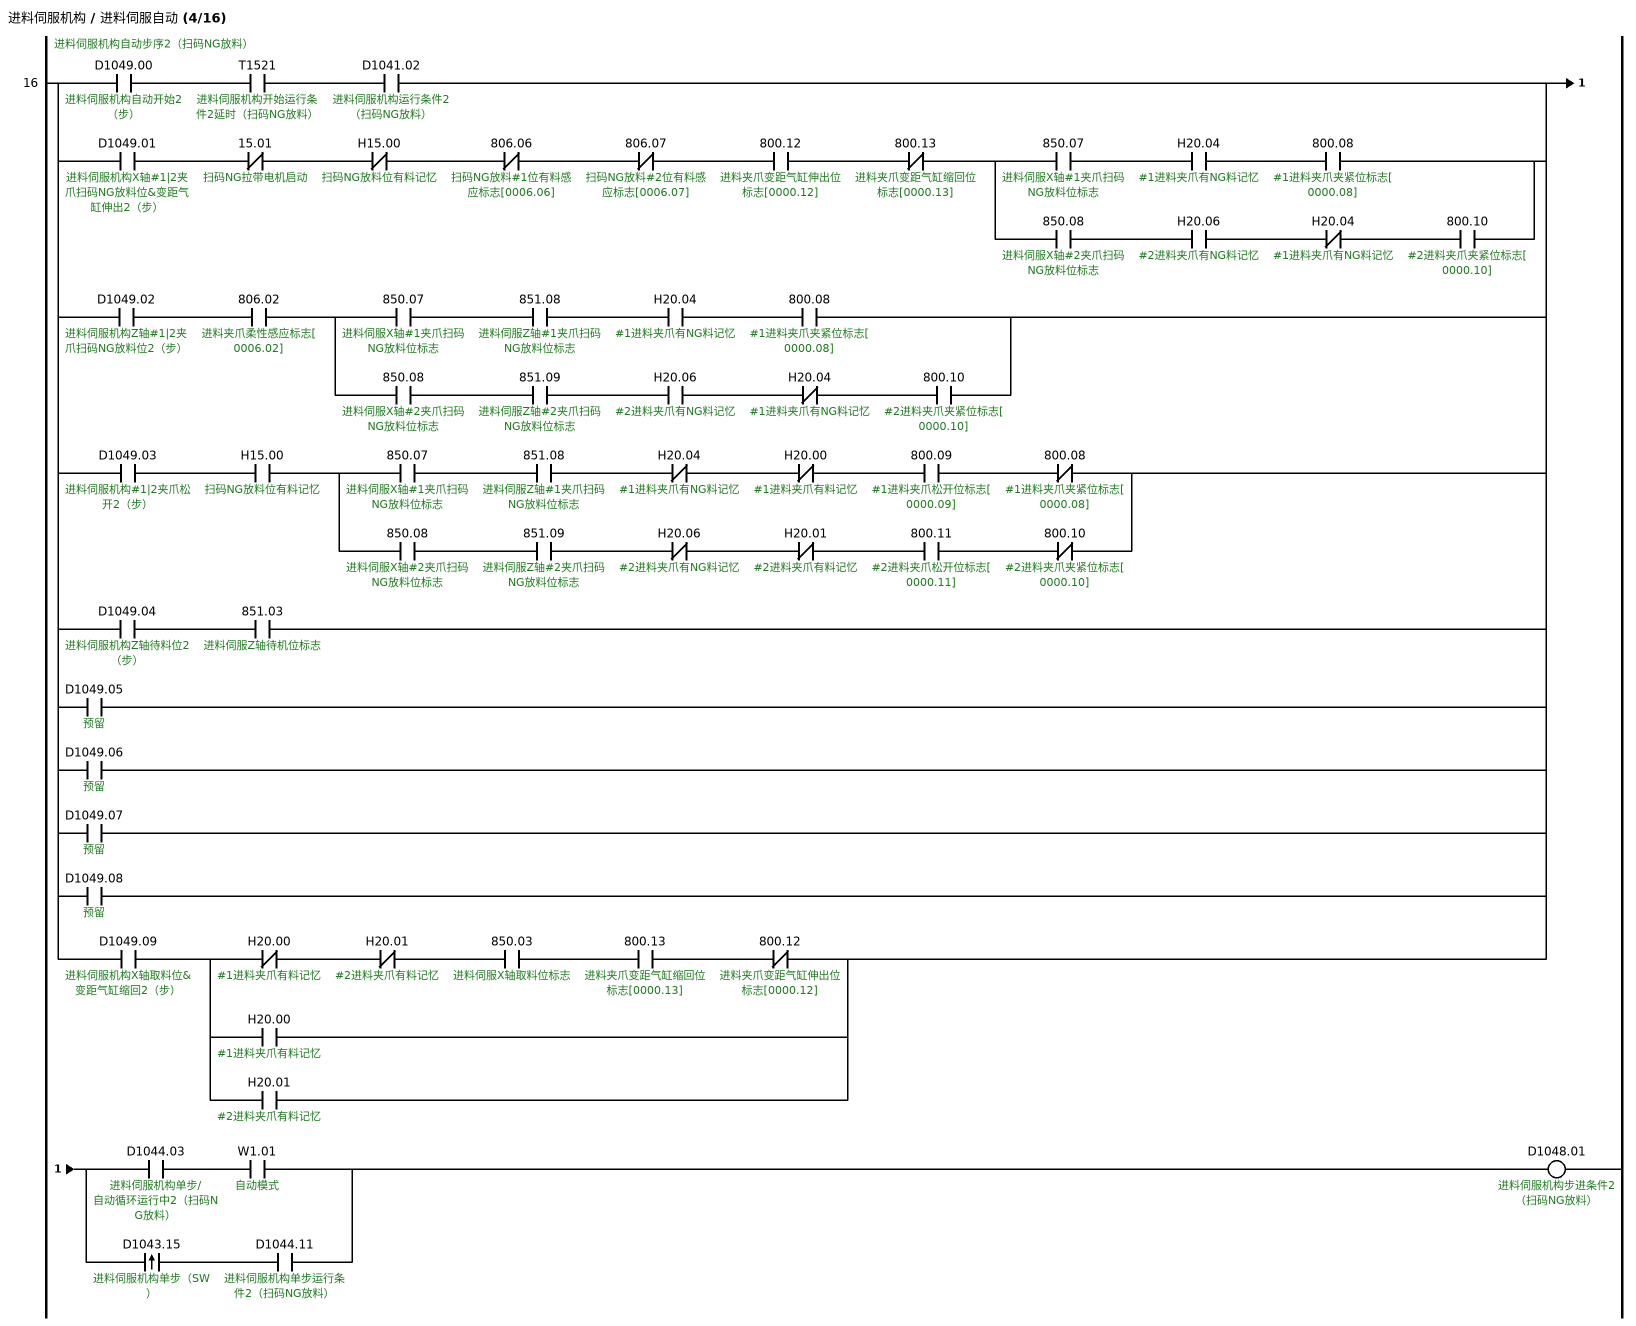
; rung 16: 进料伺服机构自动步序2（扫码NG放料）
LD D1049.00  ; 进料伺服机构自动开始2（步）
AND T1521  ; 进料伺服机构开始运行条件2延时（扫码NG放料）
AND D1041.02  ; 进料伺服机构运行条件2（扫码NG放料）
LD D1049.01  ; 进料伺服机构X轴#1|2夹爪扫码NG放料位&变距气缸伸出2（步）
ANDNOT 15.01  ; 扫码NG拉带电机启动
ANDNOT H15.00  ; 扫码NG放料位有料记忆
ANDNOT 806.06  ; 扫码NG放料#1位有料感应标志[0006.06]
ANDNOT 806.07  ; 扫码NG放料#2位有料感应标志[0006.07]
AND 800.12  ; 进料夹爪变距气缸伸出位标志[0000.12]
ANDNOT 800.13  ; 进料夹爪变距气缸缩回位标志[0000.13]
LD 850.07  ; 进料伺服X轴#1夹爪扫码NG放料位标志
AND H20.04  ; #1进料夹爪有NG料记忆
AND 800.08  ; #1进料夹爪夹紧位标志[0000.08]
LD 850.08  ; 进料伺服X轴#2夹爪扫码NG放料位标志
AND H20.06  ; #2进料夹爪有NG料记忆
ANDNOT H20.04  ; #1进料夹爪有NG料记忆
AND 800.10  ; #2进料夹爪夹紧位标志[0000.10]
ORLD
ANDLD
ORLD
LD D1049.02  ; 进料伺服机构Z轴#1|2夹爪扫码NG放料位2（步）
AND 806.02  ; 进料夹爪柔性感应标志[0006.02]
LD 850.07  ; 进料伺服X轴#1夹爪扫码NG放料位标志
AND 851.08  ; 进料伺服Z轴#1夹爪扫码NG放料位标志
AND H20.04  ; #1进料夹爪有NG料记忆
AND 800.08  ; #1进料夹爪夹紧位标志[0000.08]
LD 850.08  ; 进料伺服X轴#2夹爪扫码NG放料位标志
AND 851.09  ; 进料伺服Z轴#2夹爪扫码NG放料位标志
AND H20.06  ; #2进料夹爪有NG料记忆
ANDNOT H20.04  ; #1进料夹爪有NG料记忆
AND 800.10  ; #2进料夹爪夹紧位标志[0000.10]
ORLD
ANDLD
ORLD
LD D1049.03  ; 进料伺服机构#1|2夹爪松开2（步）
AND H15.00  ; 扫码NG放料位有料记忆
LD 850.07  ; 进料伺服X轴#1夹爪扫码NG放料位标志
AND 851.08  ; 进料伺服Z轴#1夹爪扫码NG放料位标志
ANDNOT H20.04  ; #1进料夹爪有NG料记忆
ANDNOT H20.00  ; #1进料夹爪有料记忆
AND 800.09  ; #1进料夹爪松开位标志[0000.09]
ANDNOT 800.08  ; #1进料夹爪夹紧位标志[0000.08]
LD 850.08  ; 进料伺服X轴#2夹爪扫码NG放料位标志
AND 851.09  ; 进料伺服Z轴#2夹爪扫码NG放料位标志
ANDNOT H20.06  ; #2进料夹爪有NG料记忆
ANDNOT H20.01  ; #2进料夹爪有料记忆
AND 800.11  ; #2进料夹爪松开位标志[0000.11]
ANDNOT 800.10  ; #2进料夹爪夹紧位标志[0000.10]
ORLD
ANDLD
ORLD
LD D1049.04  ; 进料伺服机构Z轴待料位2（步）
AND 851.03  ; 进料伺服Z轴待机位标志
ORLD
OR D1049.05  ; 预留
OR D1049.06  ; 预留
OR D1049.07  ; 预留
OR D1049.08  ; 预留
LD D1049.09  ; 进料伺服机构X轴取料位&变距气缸缩回2（步）
LDNOT H20.00  ; #1进料夹爪有料记忆
ANDNOT H20.01  ; #2进料夹爪有料记忆
AND 850.03  ; 进料伺服X轴取料位标志
AND 800.13  ; 进料夹爪变距气缸缩回位标志[0000.13]
ANDNOT 800.12  ; 进料夹爪变距气缸伸出位标志[0000.12]
OR H20.00  ; #1进料夹爪有料记忆
OR H20.01  ; #2进料夹爪有料记忆
ANDLD
ORLD
LD D1044.03  ; 进料伺服机构单步/自动循环运行中2（扫码NG放料）
AND W1.01  ; 自动模式
@LD D1043.15  ; 进料伺服机构单步（SW）
AND D1044.11  ; 进料伺服机构单步运行条件2（扫码NG放料）
ORLD
ANDLD
OUT D1048.01  ; 进料伺服机构步进条件2（扫码NG放料）

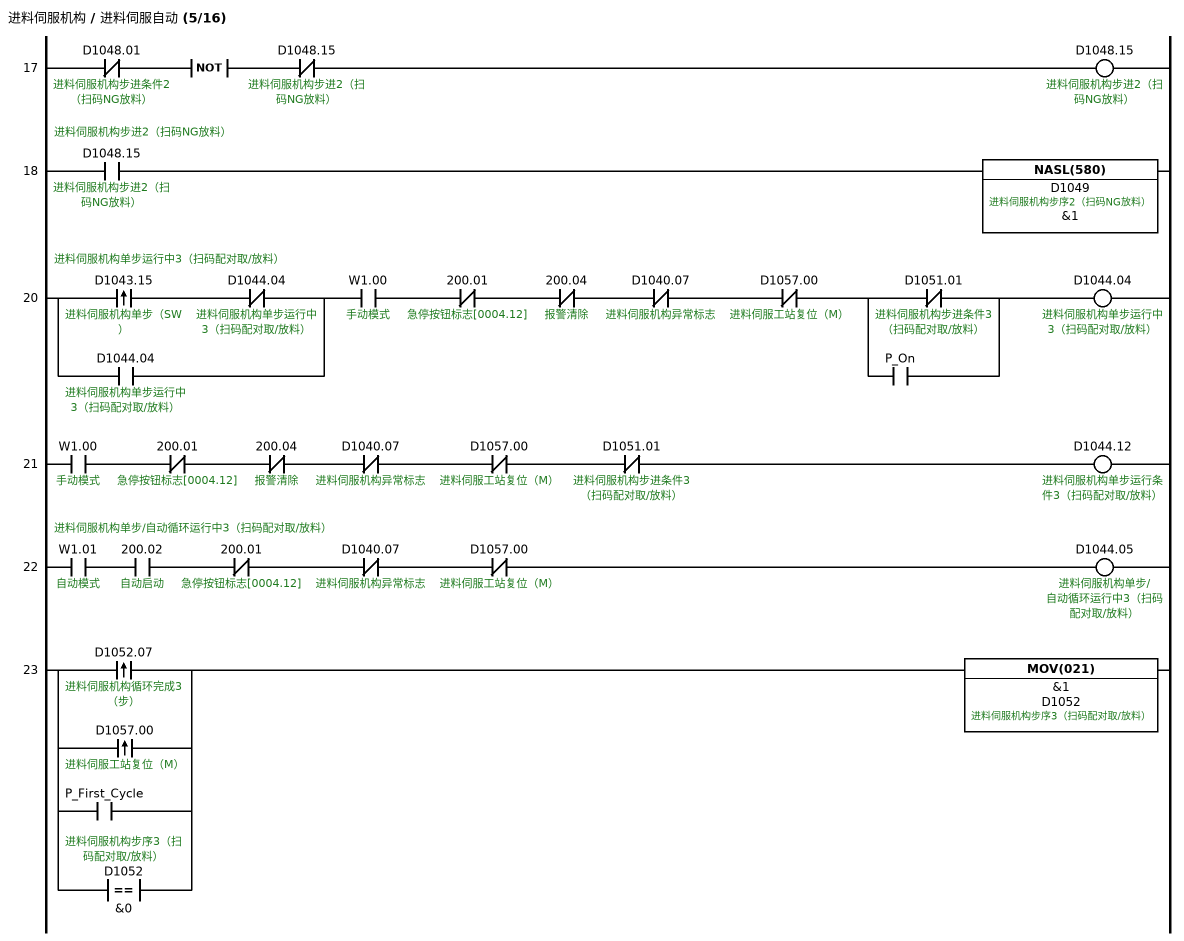
; rung 17
LDNOT D1048.01  ; 进料伺服机构步进条件2（扫码NG放料）
NOT(520)
ANDNOT D1048.15  ; 进料伺服机构步进2（扫码NG放料）
OUT D1048.15  ; 进料伺服机构步进2（扫码NG放料）
; rung 18: 进料伺服机构步进2（扫码NG放料）
LD D1048.15  ; 进料伺服机构步进2（扫码NG放料）
NASL(580) D1049 &1  ; 进料伺服机构步序2（扫码NG放料）
; rung 19: 进料伺服机构步序跳转程序2（扫码NG放料）
; rung 20: 进料伺服机构单步运行中3（扫码配对取/放料）
@LD D1043.15  ; 进料伺服机构单步（SW）
ANDNOT D1044.04  ; 进料伺服机构单步运行中3（扫码配对取/放料）
OR D1044.04  ; 进料伺服机构单步运行中3（扫码配对取/放料）
AND W1.00  ; 手动模式
ANDNOT 200.01  ; 急停按钮标志[0004.12]
ANDNOT 200.04  ; 报警清除
ANDNOT D1040.07  ; 进料伺服机构异常标志
ANDNOT D1057.00  ; 进料伺服工站复位（M）
LDNOT D1051.01  ; 进料伺服机构步进条件3（扫码配对取/放料）
OR P_On
ANDLD
OUT D1044.04  ; 进料伺服机构单步运行中3（扫码配对取/放料）
; rung 21
LD W1.00  ; 手动模式
ANDNOT 200.01  ; 急停按钮标志[0004.12]
ANDNOT 200.04  ; 报警清除
ANDNOT D1040.07  ; 进料伺服机构异常标志
ANDNOT D1057.00  ; 进料伺服工站复位（M）
ANDNOT D1051.01  ; 进料伺服机构步进条件3（扫码配对取/放料）
OUT D1044.12  ; 进料伺服机构单步运行条件3（扫码配对取/放料）
; rung 22: 进料伺服机构单步/自动循环运行中3（扫码配对取/放料）
LD W1.01  ; 自动模式
AND 200.02  ; 自动启动
ANDNOT 200.01  ; 急停按钮标志[0004.12]
ANDNOT D1040.07  ; 进料伺服机构异常标志
ANDNOT D1057.00  ; 进料伺服工站复位（M）
OUT D1044.05  ; 进料伺服机构单步/自动循环运行中3（扫码配对取/放料）
; rung 23
@LD D1052.07  ; 进料伺服机构循环完成3（步）
@OR D1057.00  ; 进料伺服工站复位（M）
OR P_First_Cycle
OR=(300) D1052 &0  ; 进料伺服机构步序3（扫码配对取/放料）
MOV(021) &1 D1052  ; 进料伺服机构步序3（扫码配对取/放料）

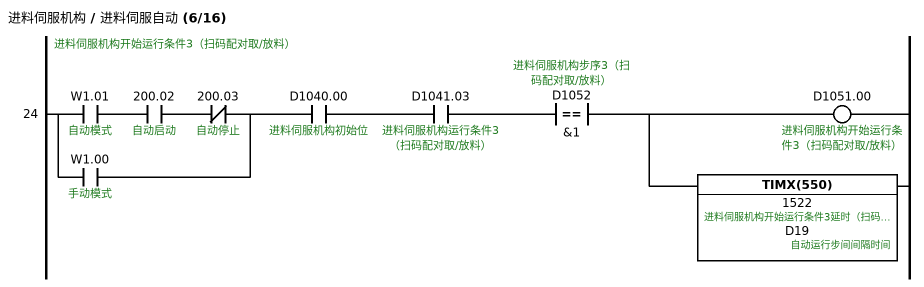
; rung 24: 进料伺服机构开始运行条件3（扫码配对取/放料）
LD W1.01  ; 自动模式
AND 200.02  ; 自动启动
ANDNOT 200.03  ; 自动停止
OR W1.00  ; 手动模式
AND D1040.00  ; 进料伺服机构初始位
AND D1041.03  ; 进料伺服机构运行条件3（扫码配对取/放料）
AND=(300) D1052 &1  ; 进料伺服机构步序3（扫码配对取/放料）
OUT D1051.00  ; 进料伺服机构开始运行条件3（扫码配对取/放料）
TIMX(550) 1522 D19  ; 自动运行步间间隔时间, 进料伺服机构开始运行条件3延时（扫码配对取/放料）

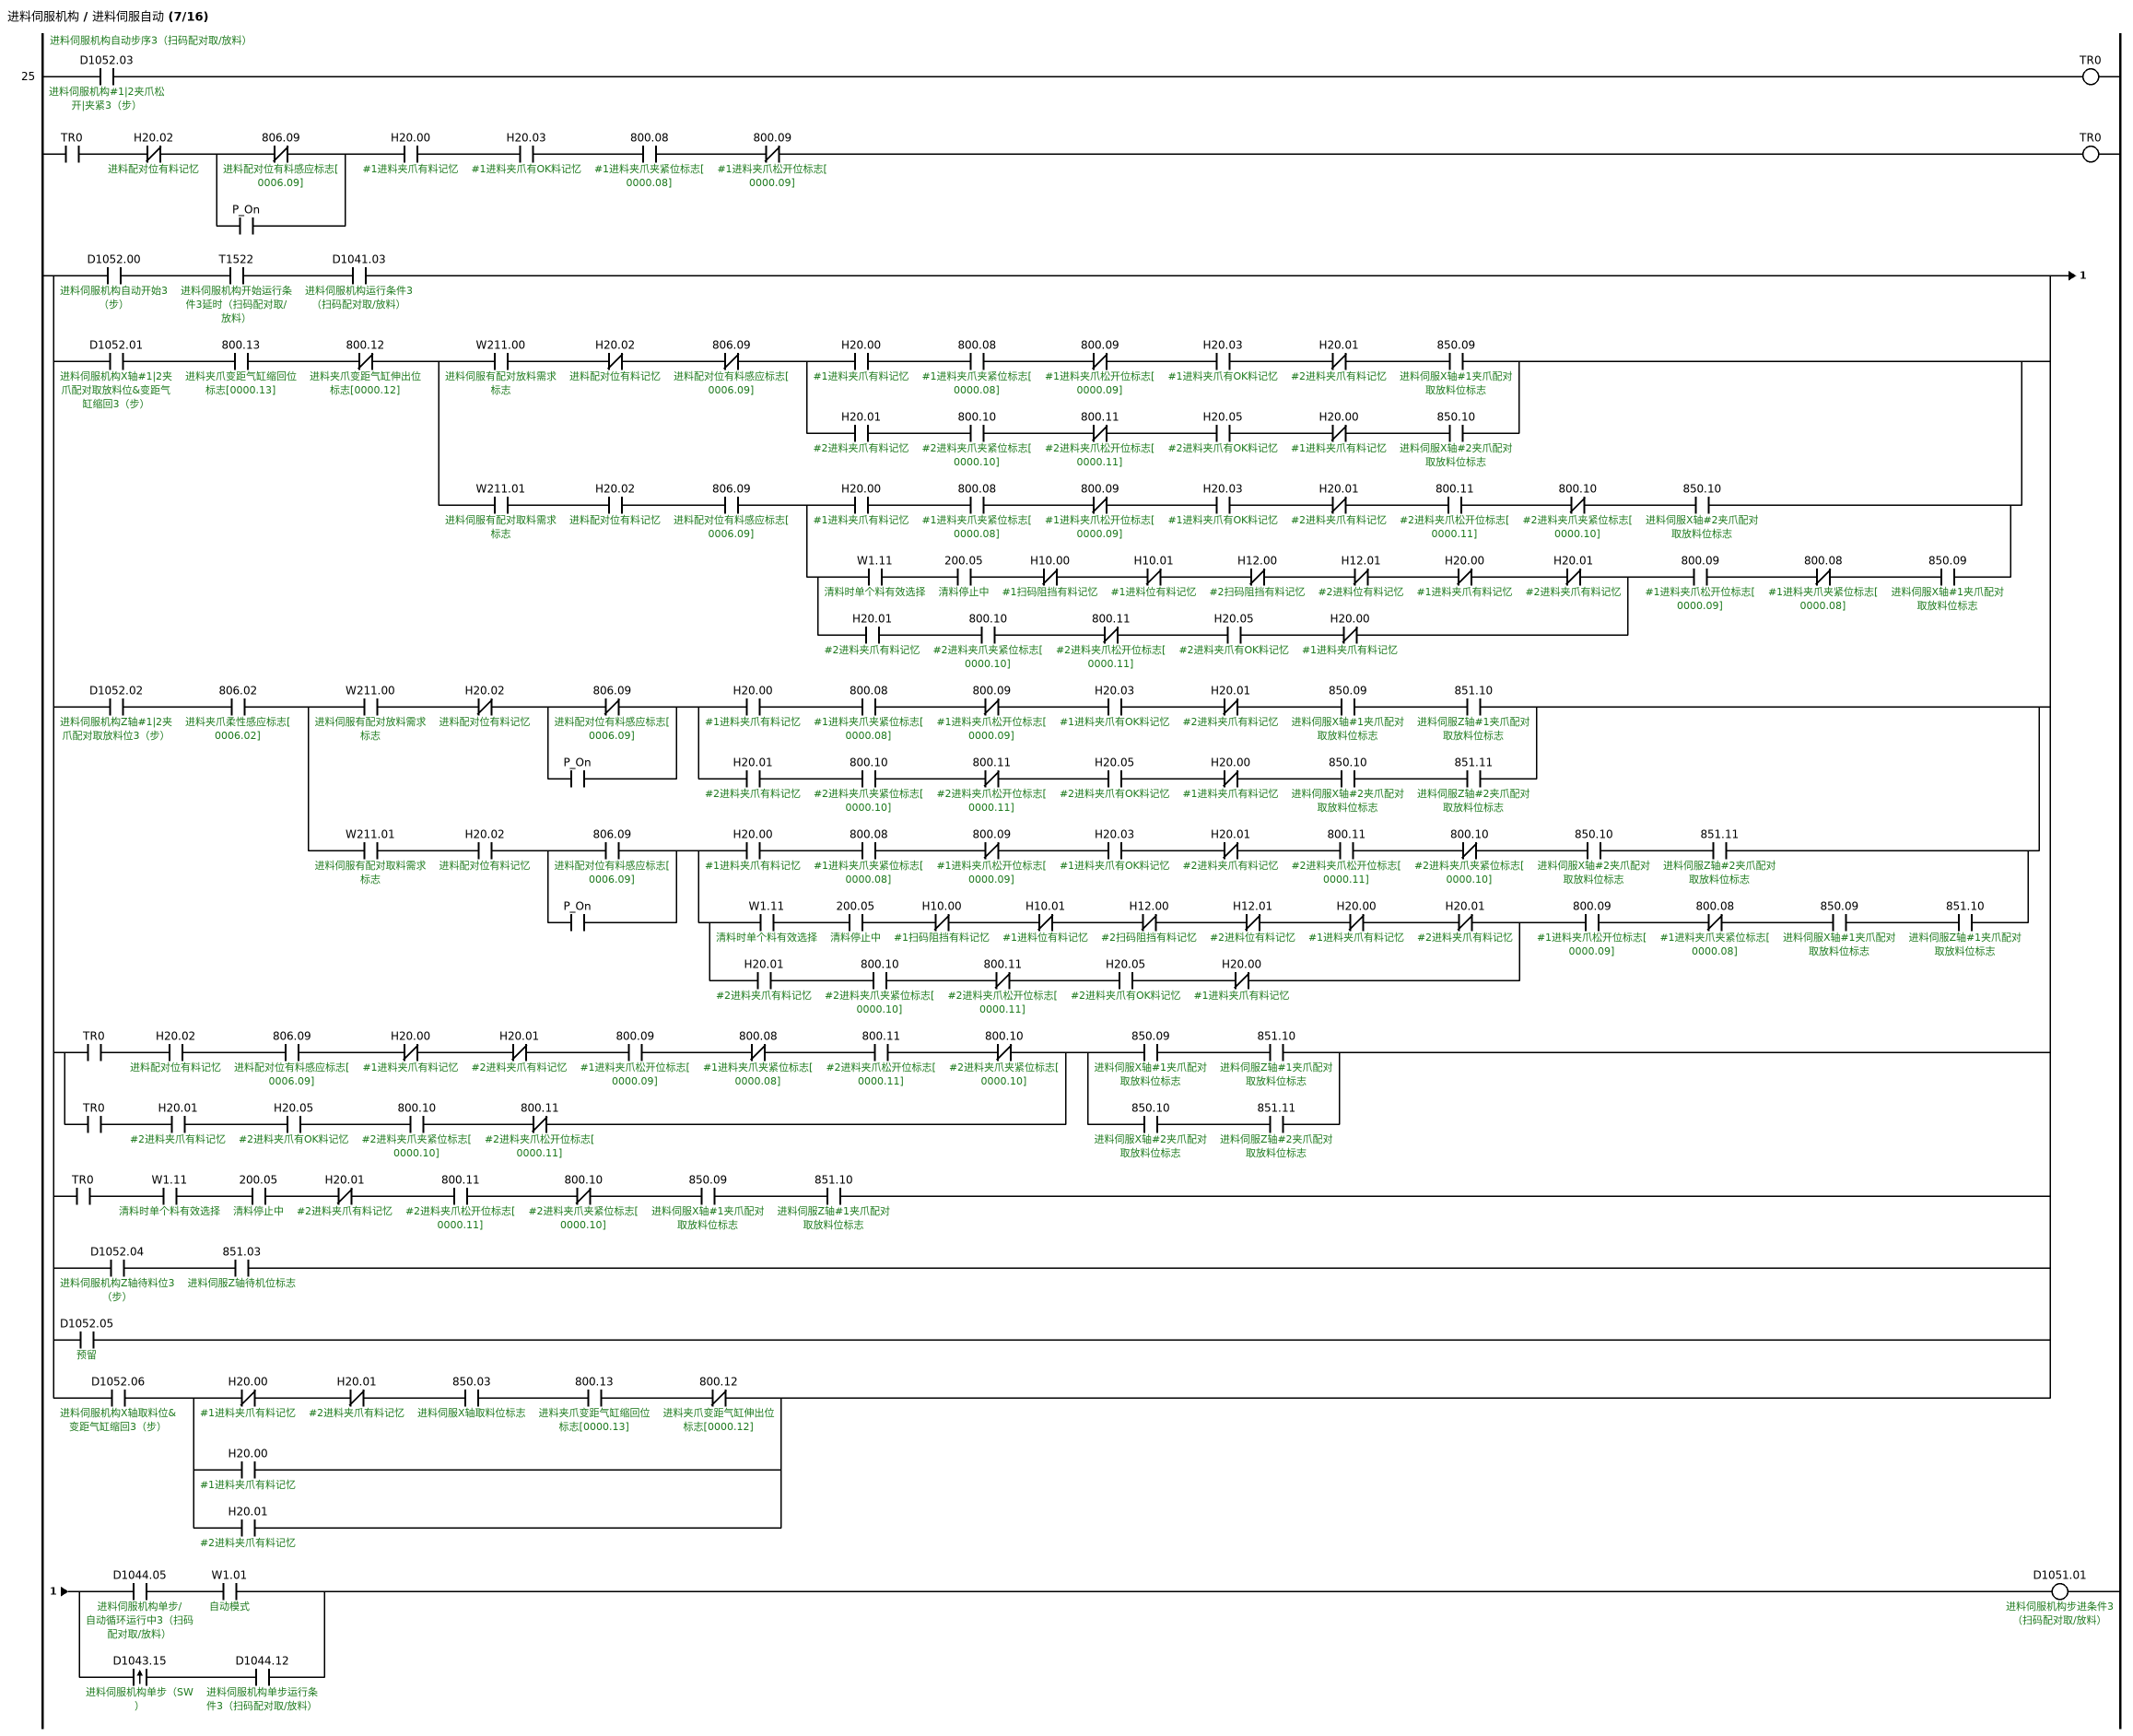
; rung 25: 进料伺服机构自动步序3（扫码配对取/放料）
LD D1052.00  ; 进料伺服机构自动开始3（步）
AND T1522  ; 进料伺服机构开始运行条件3延时（扫码配对取/放料）
AND D1041.03  ; 进料伺服机构运行条件3（扫码配对取/放料）
LD D1052.01  ; 进料伺服机构X轴#1|2夹爪配对取放料位&变距气缸缩回3（步）
AND 800.13  ; 进料夹爪变距气缸缩回位标志[0000.13]
ANDNOT 800.12  ; 进料夹爪变距气缸伸出位标志[0000.12]
LD W211.00  ; 进料伺服有配对放料需求标志
ANDNOT H20.02  ; 进料配对位有料记忆
ANDNOT 806.09  ; 进料配对位有料感应标志[0006.09]
LD H20.00  ; #1进料夹爪有料记忆
AND 800.08  ; #1进料夹爪夹紧位标志[0000.08]
ANDNOT 800.09  ; #1进料夹爪松开位标志[0000.09]
AND H20.03  ; #1进料夹爪有OK料记忆
ANDNOT H20.01  ; #2进料夹爪有料记忆
AND 850.09  ; 进料伺服X轴#1夹爪配对取放料位标志
LD H20.01  ; #2进料夹爪有料记忆
AND 800.10  ; #2进料夹爪夹紧位标志[0000.10]
ANDNOT 800.11  ; #2进料夹爪松开位标志[0000.11]
AND H20.05  ; #2进料夹爪有OK料记忆
ANDNOT H20.00  ; #1进料夹爪有料记忆
AND 850.10  ; 进料伺服X轴#2夹爪配对取放料位标志
ORLD
ANDLD
LD W211.01  ; 进料伺服有配对取料需求标志
AND H20.02  ; 进料配对位有料记忆
AND 806.09  ; 进料配对位有料感应标志[0006.09]
LD H20.00  ; #1进料夹爪有料记忆
AND 800.08  ; #1进料夹爪夹紧位标志[0000.08]
ANDNOT 800.09  ; #1进料夹爪松开位标志[0000.09]
AND H20.03  ; #1进料夹爪有OK料记忆
ANDNOT H20.01  ; #2进料夹爪有料记忆
AND 800.11  ; #2进料夹爪松开位标志[0000.11]
ANDNOT 800.10  ; #2进料夹爪夹紧位标志[0000.10]
AND 850.10  ; 进料伺服X轴#2夹爪配对取放料位标志
LD W1.11  ; 清料时单个料有效选择
AND 200.05  ; 清料停止中  // 清料时，如进料端只有配对缓存有料，其它没料，则#1进料夹爪优先取料！！
ANDNOT H10.00  ; #1扫码阻挡有料记忆
ANDNOT H10.01  ; #1进料位有料记忆
ANDNOT H12.00  ; #2扫码阻挡有料记忆
ANDNOT H12.01  ; #2进料位有料记忆
ANDNOT H20.00  ; #1进料夹爪有料记忆
ANDNOT H20.01  ; #2进料夹爪有料记忆
LD H20.01  ; #2进料夹爪有料记忆
AND 800.10  ; #2进料夹爪夹紧位标志[0000.10]
ANDNOT 800.11  ; #2进料夹爪松开位标志[0000.11]
AND H20.05  ; #2进料夹爪有OK料记忆
ANDNOT H20.00  ; #1进料夹爪有料记忆
ORLD
AND 800.09  ; #1进料夹爪松开位标志[0000.09]
ANDNOT 800.08  ; #1进料夹爪夹紧位标志[0000.08]
AND 850.09  ; 进料伺服X轴#1夹爪配对取放料位标志
ORLD
ANDLD
ORLD
ANDLD
ORLD
LD D1052.02  ; 进料伺服机构Z轴#1|2夹爪配对取放料位3（步）
AND 806.02  ; 进料夹爪柔性感应标志[0006.02]
LD W211.00  ; 进料伺服有配对放料需求标志
ANDNOT H20.02  ; 进料配对位有料记忆
LDNOT 806.09  ; 进料配对位有料感应标志[0006.09]
OR P_On
ANDLD
LD H20.00  ; #1进料夹爪有料记忆
AND 800.08  ; #1进料夹爪夹紧位标志[0000.08]
ANDNOT 800.09  ; #1进料夹爪松开位标志[0000.09]
AND H20.03  ; #1进料夹爪有OK料记忆
ANDNOT H20.01  ; #2进料夹爪有料记忆
AND 850.09  ; 进料伺服X轴#1夹爪配对取放料位标志
AND 851.10  ; 进料伺服Z轴#1夹爪配对取放料位标志
LD H20.01  ; #2进料夹爪有料记忆
AND 800.10  ; #2进料夹爪夹紧位标志[0000.10]
ANDNOT 800.11  ; #2进料夹爪松开位标志[0000.11]
AND H20.05  ; #2进料夹爪有OK料记忆
ANDNOT H20.00  ; #1进料夹爪有料记忆
AND 850.10  ; 进料伺服X轴#2夹爪配对取放料位标志
AND 851.11  ; 进料伺服Z轴#2夹爪配对取放料位标志
ORLD
ANDLD
LD W211.01  ; 进料伺服有配对取料需求标志
AND H20.02  ; 进料配对位有料记忆
LD 806.09  ; 进料配对位有料感应标志[0006.09]
OR P_On
ANDLD
LD H20.00  ; #1进料夹爪有料记忆
AND 800.08  ; #1进料夹爪夹紧位标志[0000.08]
ANDNOT 800.09  ; #1进料夹爪松开位标志[0000.09]
AND H20.03  ; #1进料夹爪有OK料记忆
ANDNOT H20.01  ; #2进料夹爪有料记忆
AND 800.11  ; #2进料夹爪松开位标志[0000.11]
ANDNOT 800.10  ; #2进料夹爪夹紧位标志[0000.10]
AND 850.10  ; 进料伺服X轴#2夹爪配对取放料位标志
AND 851.11  ; 进料伺服Z轴#2夹爪配对取放料位标志
LD W1.11  ; 清料时单个料有效选择
AND 200.05  ; 清料停止中
ANDNOT H10.00  ; #1扫码阻挡有料记忆
ANDNOT H10.01  ; #1进料位有料记忆
ANDNOT H12.00  ; #2扫码阻挡有料记忆
ANDNOT H12.01  ; #2进料位有料记忆
ANDNOT H20.00  ; #1进料夹爪有料记忆
ANDNOT H20.01  ; #2进料夹爪有料记忆
LD H20.01  ; #2进料夹爪有料记忆
AND 800.10  ; #2进料夹爪夹紧位标志[0000.10]
ANDNOT 800.11  ; #2进料夹爪松开位标志[0000.11]
AND H20.05  ; #2进料夹爪有OK料记忆
ANDNOT H20.00  ; #1进料夹爪有料记忆
ORLD
AND 800.09  ; #1进料夹爪松开位标志[0000.09]
ANDNOT 800.08  ; #1进料夹爪夹紧位标志[0000.08]
AND 850.09  ; 进料伺服X轴#1夹爪配对取放料位标志
AND 851.10  ; 进料伺服Z轴#1夹爪配对取放料位标志
ORLD
ANDLD
ORLD
ANDLD
ORLD
LD D1052.03  ; 进料伺服机构#1|2夹爪松开|夹紧3（步）
OUT TR0
AND H20.02  ; 进料配对位有料记忆  // 放料
AND 806.09  ; 进料配对位有料感应标志[0006.09]
ANDNOT H20.00  ; #1进料夹爪有料记忆
ANDNOT H20.01  ; #2进料夹爪有料记忆
AND 800.09  ; #1进料夹爪松开位标志[0000.09]
ANDNOT 800.08  ; #1进料夹爪夹紧位标志[0000.08]
AND 800.11  ; #2进料夹爪松开位标志[0000.11]
ANDNOT 800.10  ; #2进料夹爪夹紧位标志[0000.10]
LD TR0
ANDNOT H20.02  ; 进料配对位有料记忆  // 取料
LDNOT 806.09  ; 进料配对位有料感应标志[0006.09]
OR P_On
ANDLD
AND H20.00  ; #1进料夹爪有料记忆
AND H20.03  ; #1进料夹爪有OK料记忆
AND 800.08  ; #1进料夹爪夹紧位标志[0000.08]
ANDNOT 800.09  ; #1进料夹爪松开位标志[0000.09]
OUT TR0
AND H20.01  ; #2进料夹爪有料记忆
AND H20.05  ; #2进料夹爪有OK料记忆
AND 800.10  ; #2进料夹爪夹紧位标志[0000.10]
ANDNOT 800.11  ; #2进料夹爪松开位标志[0000.11]
ORLD
LD 850.09  ; 进料伺服X轴#1夹爪配对取放料位标志
AND 851.10  ; 进料伺服Z轴#1夹爪配对取放料位标志
LD 850.10  ; 进料伺服X轴#2夹爪配对取放料位标志
AND 851.11  ; 进料伺服Z轴#2夹爪配对取放料位标志
ORLD
ANDLD
ORLD
LD TR0
AND W1.11  ; 清料时单个料有效选择
AND 200.05  ; 清料停止中
ANDNOT H20.01  ; #2进料夹爪有料记忆
AND 800.11  ; #2进料夹爪松开位标志[0000.11]
ANDNOT 800.10  ; #2进料夹爪夹紧位标志[0000.10]
AND 850.09  ; 进料伺服X轴#1夹爪配对取放料位标志
AND 851.10  ; 进料伺服Z轴#1夹爪配对取放料位标志
LD D1052.04  ; 进料伺服机构Z轴待料位3（步）
AND 851.03  ; 进料伺服Z轴待机位标志
OR D1052.05  ; 预留
LD D1052.06  ; 进料伺服机构X轴取料位&变距气缸缩回3（步）
LDNOT H20.00  ; #1进料夹爪有料记忆
ANDNOT H20.01  ; #2进料夹爪有料记忆
AND 850.03  ; 进料伺服X轴取料位标志
AND 800.13  ; 进料夹爪变距气缸缩回位标志[0000.13]
ANDNOT 800.12  ; 进料夹爪变距气缸伸出位标志[0000.12]
OR H20.00  ; #1进料夹爪有料记忆
OR H20.01  ; #2进料夹爪有料记忆
ANDLD
ORLD
ORLD
ORLD
LD D1044.05  ; 进料伺服机构单步/自动循环运行中3（扫码配对取/放料）
AND W1.01  ; 自动模式
@LD D1043.15  ; 进料伺服机构单步（SW）
AND D1044.12  ; 进料伺服机构单步运行条件3（扫码配对取/放料）
ORLD
ANDLD
OUT D1051.01  ; 进料伺服机构步进条件3（扫码配对取/放料）

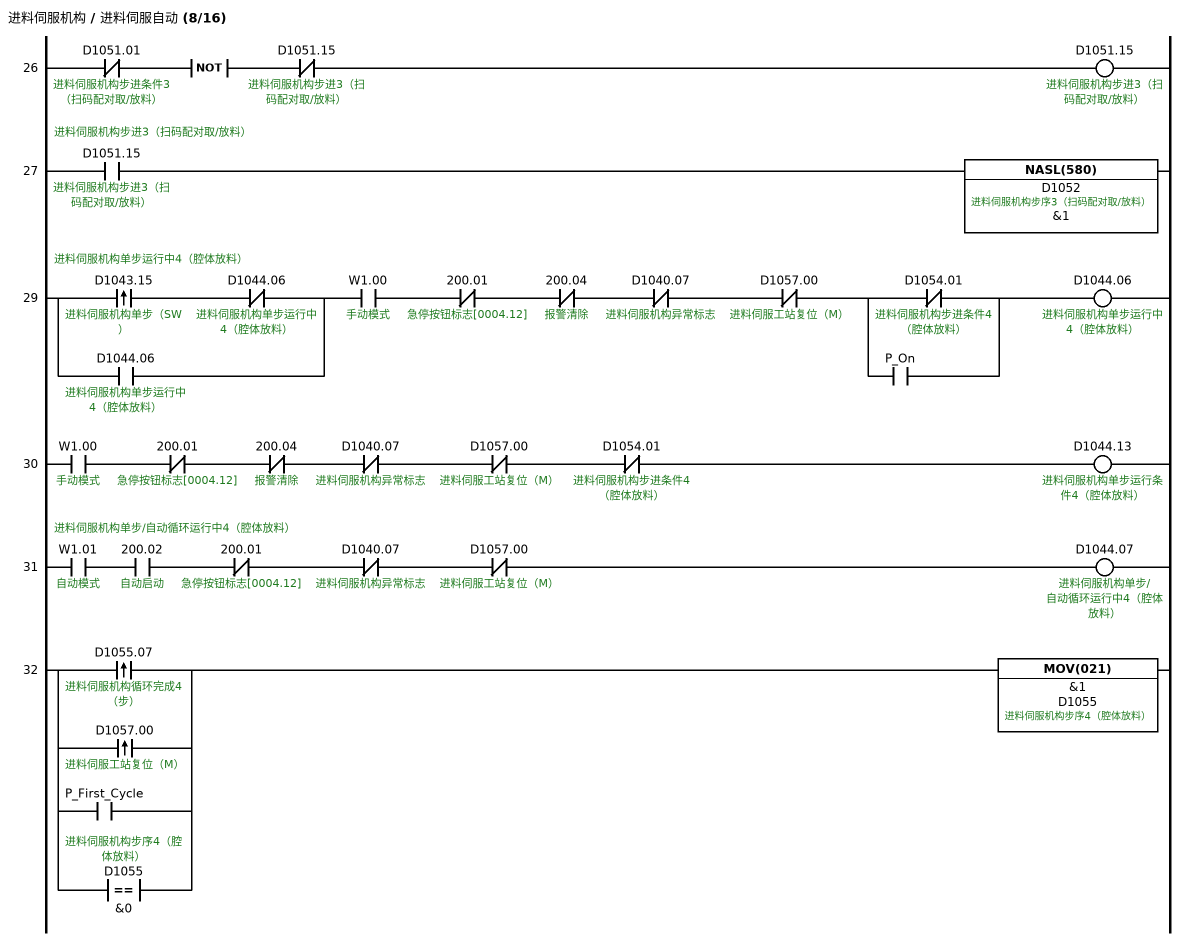
; rung 26
LDNOT D1051.01  ; 进料伺服机构步进条件3（扫码配对取/放料）
NOT(520)
ANDNOT D1051.15  ; 进料伺服机构步进3（扫码配对取/放料）
OUT D1051.15  ; 进料伺服机构步进3（扫码配对取/放料）
; rung 27: 进料伺服机构步进3（扫码配对取/放料）
LD D1051.15  ; 进料伺服机构步进3（扫码配对取/放料）
NASL(580) D1052 &1  ; 进料伺服机构步序3（扫码配对取/放料）
; rung 28: 进料伺服机构步序跳转程序3（扫码配对取/放料）
; rung 29: 进料伺服机构单步运行中4（腔体放料）
@LD D1043.15  ; 进料伺服机构单步（SW）
ANDNOT D1044.06  ; 进料伺服机构单步运行中4（腔体放料）
OR D1044.06  ; 进料伺服机构单步运行中4（腔体放料）
AND W1.00  ; 手动模式
ANDNOT 200.01  ; 急停按钮标志[0004.12]
ANDNOT 200.04  ; 报警清除
ANDNOT D1040.07  ; 进料伺服机构异常标志
ANDNOT D1057.00  ; 进料伺服工站复位（M）
LDNOT D1054.01  ; 进料伺服机构步进条件4（腔体放料）
OR P_On
ANDLD
OUT D1044.06  ; 进料伺服机构单步运行中4（腔体放料）
; rung 30
LD W1.00  ; 手动模式
ANDNOT 200.01  ; 急停按钮标志[0004.12]
ANDNOT 200.04  ; 报警清除
ANDNOT D1040.07  ; 进料伺服机构异常标志
ANDNOT D1057.00  ; 进料伺服工站复位（M）
ANDNOT D1054.01  ; 进料伺服机构步进条件4（腔体放料）
OUT D1044.13  ; 进料伺服机构单步运行条件4（腔体放料）
; rung 31: 进料伺服机构单步/自动循环运行中4（腔体放料）
LD W1.01  ; 自动模式
AND 200.02  ; 自动启动
ANDNOT 200.01  ; 急停按钮标志[0004.12]
ANDNOT D1040.07  ; 进料伺服机构异常标志
ANDNOT D1057.00  ; 进料伺服工站复位（M）
OUT D1044.07  ; 进料伺服机构单步/自动循环运行中4（腔体放料）
; rung 32
@LD D1055.07  ; 进料伺服机构循环完成4（步）
@OR D1057.00  ; 进料伺服工站复位（M）
OR P_First_Cycle
OR=(300) D1055 &0  ; 进料伺服机构步序4（腔体放料）
MOV(021) &1 D1055  ; 进料伺服机构步序4（腔体放料）

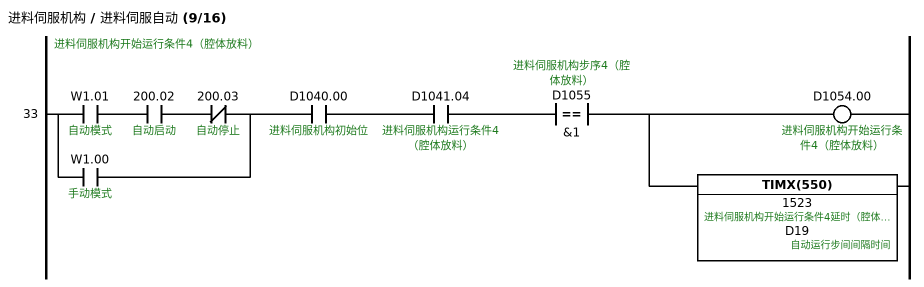
; rung 33: 进料伺服机构开始运行条件4（腔体放料）
LD W1.01  ; 自动模式
AND 200.02  ; 自动启动
ANDNOT 200.03  ; 自动停止
OR W1.00  ; 手动模式
AND D1040.00  ; 进料伺服机构初始位
AND D1041.04  ; 进料伺服机构运行条件4（腔体放料）
AND=(300) D1055 &1  ; 进料伺服机构步序4（腔体放料）
OUT D1054.00  ; 进料伺服机构开始运行条件4（腔体放料）
TIMX(550) 1523 D19  ; 自动运行步间间隔时间, 进料伺服机构开始运行条件4延时（腔体放料）

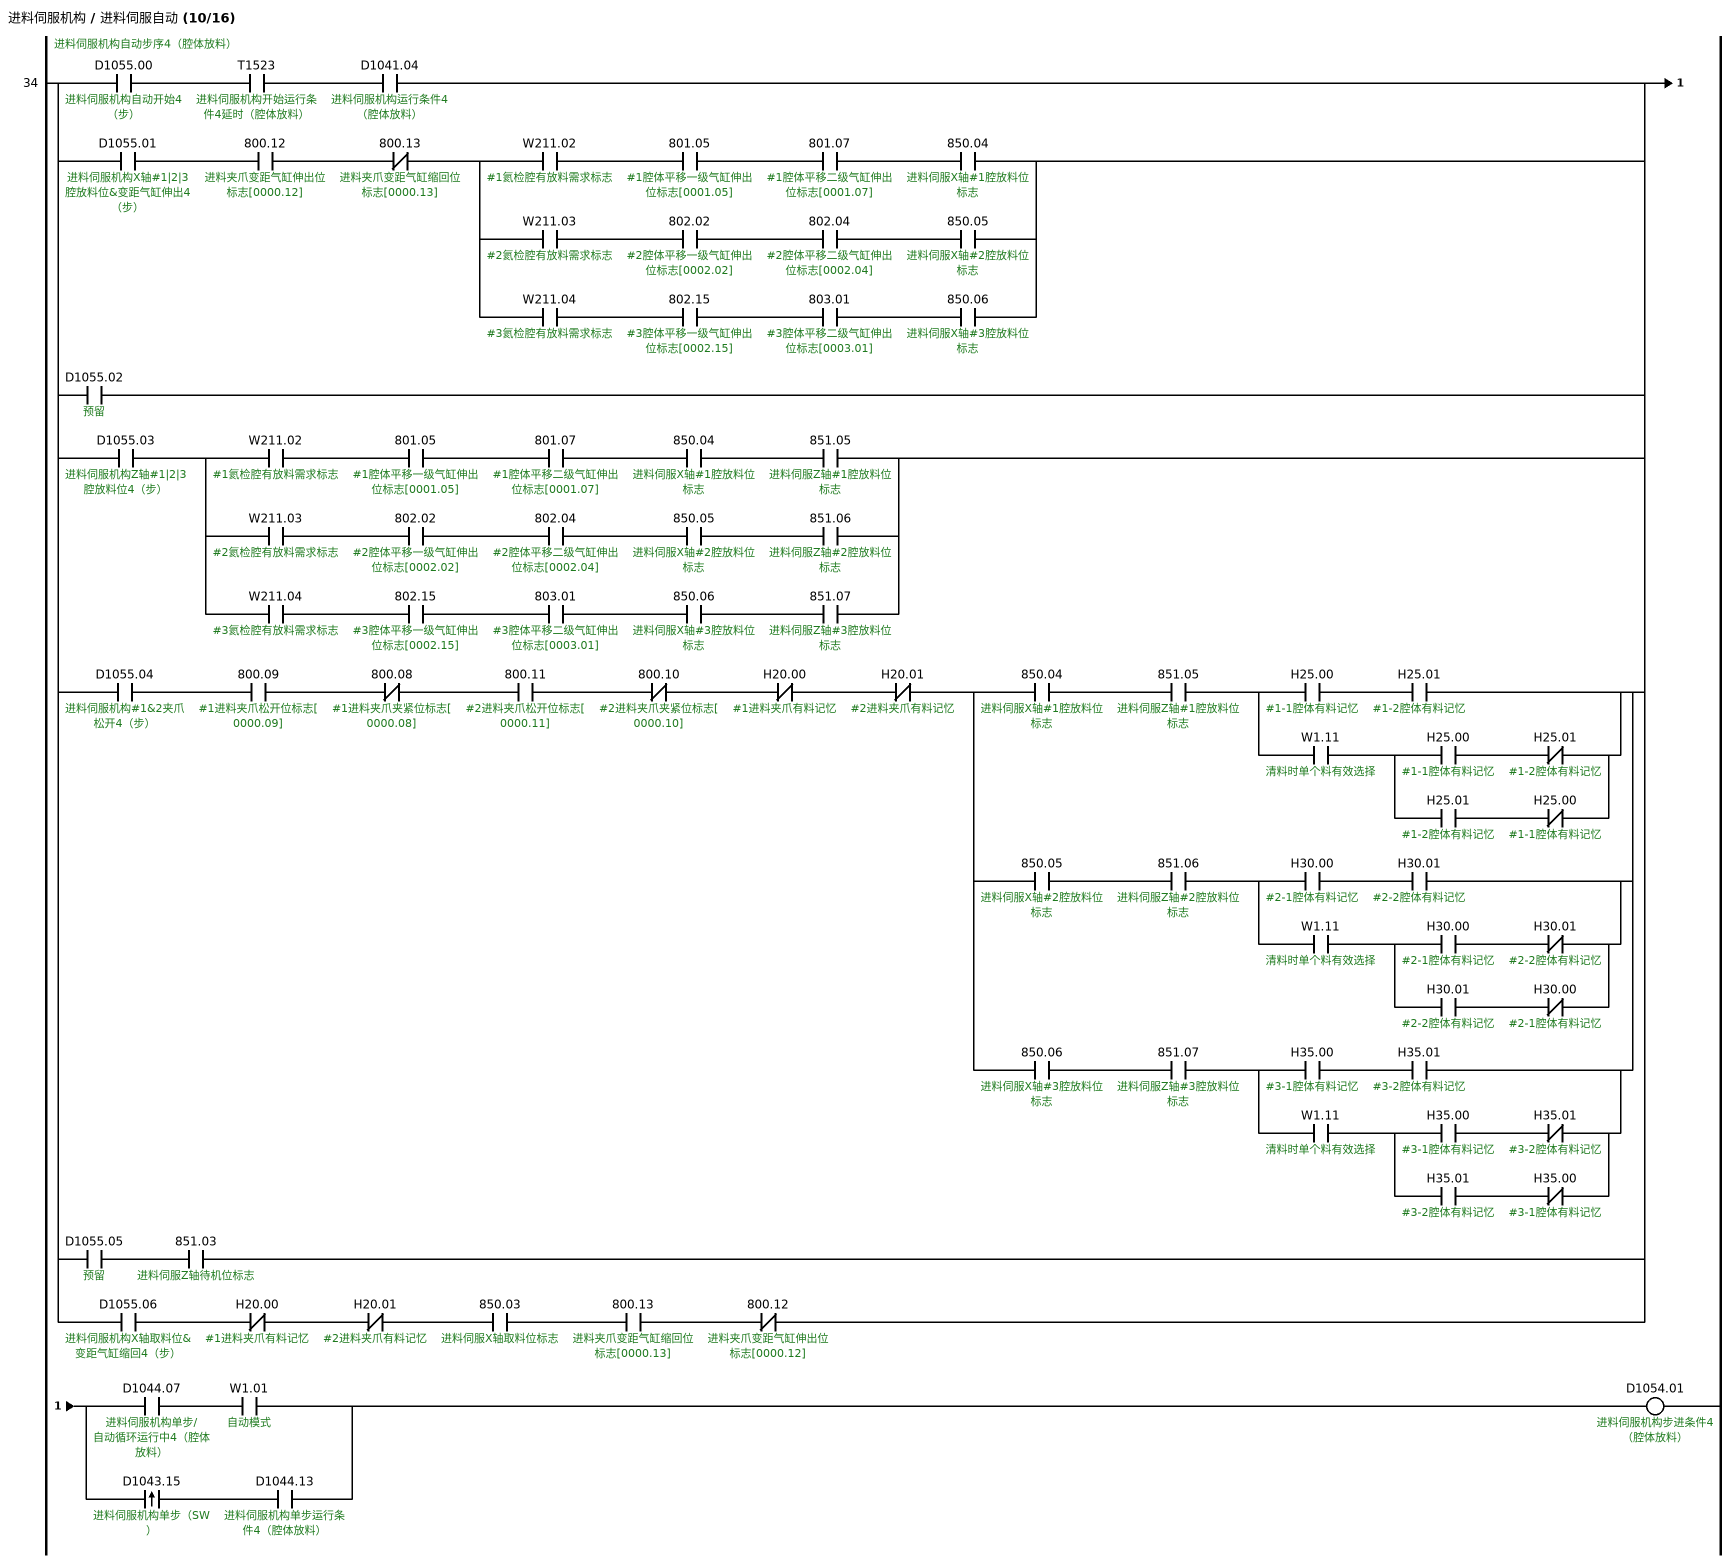
; rung 34: 进料伺服机构自动步序4（腔体放料）
LD D1055.00  ; 进料伺服机构自动开始4（步）
AND T1523  ; 进料伺服机构开始运行条件4延时（腔体放料）
AND D1041.04  ; 进料伺服机构运行条件4（腔体放料）
LD D1055.01  ; 进料伺服机构X轴#1|2|3腔放料位&变距气缸伸出4（步）
AND 800.12  ; 进料夹爪变距气缸伸出位标志[0000.12]
ANDNOT 800.13  ; 进料夹爪变距气缸缩回位标志[0000.13]
LD W211.02  ; #1氦检腔有放料需求标志
AND 801.05  ; #1腔体平移一级气缸伸出位标志[0001.05]
AND 801.07  ; #1腔体平移二级气缸伸出位标志[0001.07]
AND 850.04  ; 进料伺服X轴#1腔放料位标志
LD W211.03  ; #2氦检腔有放料需求标志
AND 802.02  ; #2腔体平移一级气缸伸出位标志[0002.02]
AND 802.04  ; #2腔体平移二级气缸伸出位标志[0002.04]
AND 850.05  ; 进料伺服X轴#2腔放料位标志
ORLD
LD W211.04  ; #3氦检腔有放料需求标志
AND 802.15  ; #3腔体平移一级气缸伸出位标志[0002.15]
AND 803.01  ; #3腔体平移二级气缸伸出位标志[0003.01]
AND 850.06  ; 进料伺服X轴#3腔放料位标志
ORLD
ANDLD
ORLD
OR D1055.02  ; 预留
LD D1055.03  ; 进料伺服机构Z轴#1|2|3腔放料位4（步）
LD W211.02  ; #1氦检腔有放料需求标志
AND 801.05  ; #1腔体平移一级气缸伸出位标志[0001.05]
AND 801.07  ; #1腔体平移二级气缸伸出位标志[0001.07]
AND 850.04  ; 进料伺服X轴#1腔放料位标志
AND 851.05  ; 进料伺服Z轴#1腔放料位标志
LD W211.03  ; #2氦检腔有放料需求标志
AND 802.02  ; #2腔体平移一级气缸伸出位标志[0002.02]
AND 802.04  ; #2腔体平移二级气缸伸出位标志[0002.04]
AND 850.05  ; 进料伺服X轴#2腔放料位标志
AND 851.06  ; 进料伺服Z轴#2腔放料位标志
ORLD
LD W211.04  ; #3氦检腔有放料需求标志
AND 802.15  ; #3腔体平移一级气缸伸出位标志[0002.15]
AND 803.01  ; #3腔体平移二级气缸伸出位标志[0003.01]
AND 850.06  ; 进料伺服X轴#3腔放料位标志
AND 851.07  ; 进料伺服Z轴#3腔放料位标志
ORLD
ANDLD
ORLD
LD D1055.04  ; 进料伺服机构#1&2夹爪松开4（步）
AND 800.09  ; #1进料夹爪松开位标志[0000.09]
ANDNOT 800.08  ; #1进料夹爪夹紧位标志[0000.08]
AND 800.11  ; #2进料夹爪松开位标志[0000.11]
ANDNOT 800.10  ; #2进料夹爪夹紧位标志[0000.10]
ANDNOT H20.00  ; #1进料夹爪有料记忆
ANDNOT H20.01  ; #2进料夹爪有料记忆
LD 850.04  ; 进料伺服X轴#1腔放料位标志
AND 851.05  ; 进料伺服Z轴#1腔放料位标志
LD H25.00  ; #1-1腔体有料记忆
AND H25.01  ; #1-2腔体有料记忆
LD W1.11  ; 清料时单个料有效选择
LD H25.00  ; #1-1腔体有料记忆
ANDNOT H25.01  ; #1-2腔体有料记忆
LD H25.01  ; #1-2腔体有料记忆
ANDNOT H25.00  ; #1-1腔体有料记忆
ORLD
ANDLD
ORLD
ANDLD
LD 850.05  ; 进料伺服X轴#2腔放料位标志
AND 851.06  ; 进料伺服Z轴#2腔放料位标志
LD H30.00  ; #2-1腔体有料记忆
AND H30.01  ; #2-2腔体有料记忆
LD W1.11  ; 清料时单个料有效选择
LD H30.00  ; #2-1腔体有料记忆
ANDNOT H30.01  ; #2-2腔体有料记忆
LD H30.01  ; #2-2腔体有料记忆
ANDNOT H30.00  ; #2-1腔体有料记忆
ORLD
ANDLD
ORLD
ANDLD
ORLD
LD 850.06  ; 进料伺服X轴#3腔放料位标志
AND 851.07  ; 进料伺服Z轴#3腔放料位标志
LD H35.00  ; #3-1腔体有料记忆
AND H35.01  ; #3-2腔体有料记忆
LD W1.11  ; 清料时单个料有效选择
LD H35.00  ; #3-1腔体有料记忆
ANDNOT H35.01  ; #3-2腔体有料记忆
LD H35.01  ; #3-2腔体有料记忆
ANDNOT H35.00  ; #3-1腔体有料记忆
ORLD
ANDLD
ORLD
ANDLD
ORLD
ANDLD
ORLD
LD D1055.05  ; 预留
AND 851.03  ; 进料伺服Z轴待机位标志
ORLD
LD D1055.06  ; 进料伺服机构X轴取料位&变距气缸缩回4（步）
ANDNOT H20.00  ; #1进料夹爪有料记忆
ANDNOT H20.01  ; #2进料夹爪有料记忆
AND 850.03  ; 进料伺服X轴取料位标志
AND 800.13  ; 进料夹爪变距气缸缩回位标志[0000.13]
ANDNOT 800.12  ; 进料夹爪变距气缸伸出位标志[0000.12]
ORLD
LD D1044.07  ; 进料伺服机构单步/自动循环运行中4（腔体放料）
AND W1.01  ; 自动模式
@LD D1043.15  ; 进料伺服机构单步（SW）
AND D1044.13  ; 进料伺服机构单步运行条件4（腔体放料）
ORLD
ANDLD
OUT D1054.01  ; 进料伺服机构步进条件4（腔体放料）

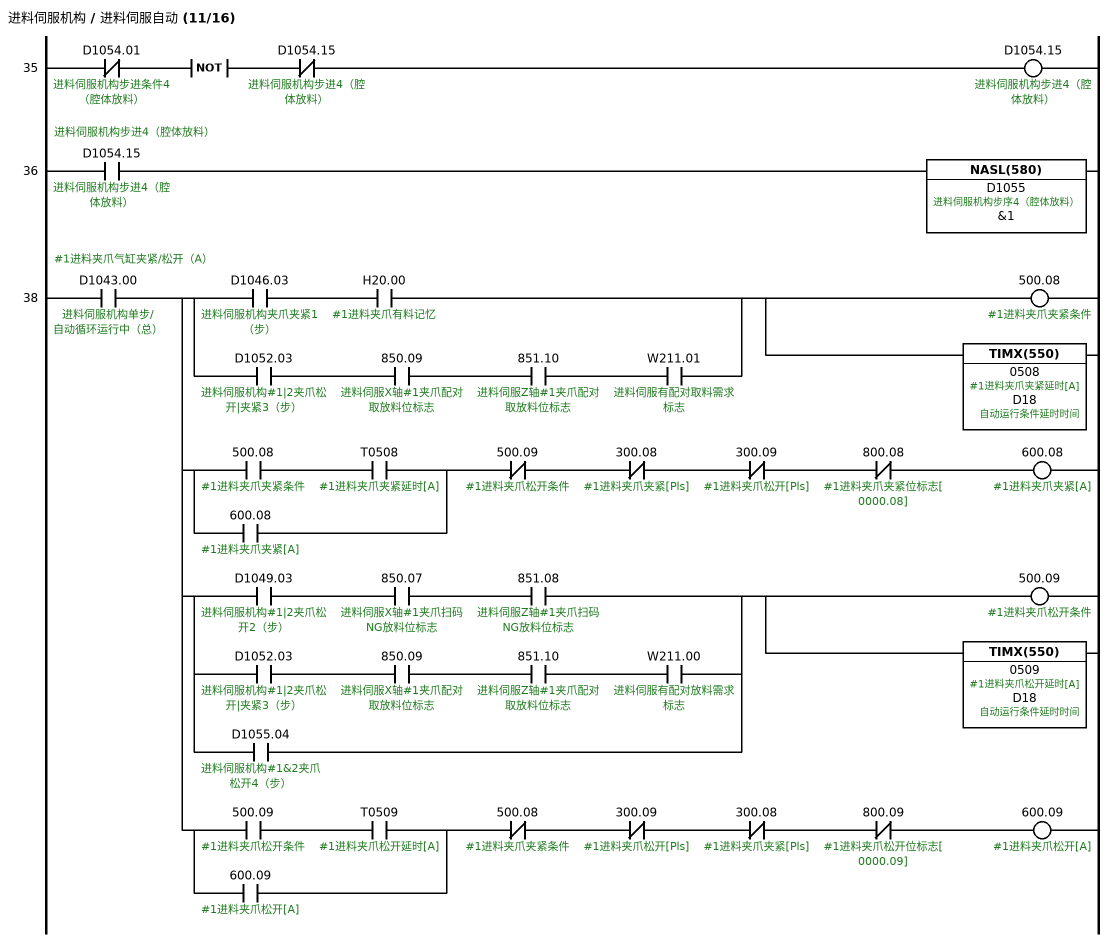
; rung 35
LDNOT D1054.01  ; 进料伺服机构步进条件4（腔体放料）
NOT(520)
ANDNOT D1054.15  ; 进料伺服机构步进4（腔体放料）
OUT D1054.15  ; 进料伺服机构步进4（腔体放料）
; rung 36: 进料伺服机构步进4（腔体放料）
LD D1054.15  ; 进料伺服机构步进4（腔体放料）
NASL(580) D1055 &1  ; 进料伺服机构步序4（腔体放料）
; rung 37: 进料伺服机构步序跳转程序4（腔体放料）
; rung 38: #1进料夹爪气缸夹紧/松开（A）
LD D1043.00  ; 进料伺服机构单步/自动循环运行中（总）
OUT TR0
LD D1046.03  ; 进料伺服机构夹爪夹紧1（步）
AND H20.00  ; #1进料夹爪有料记忆
LD D1052.03  ; 进料伺服机构#1|2夹爪松开|夹紧3（步）
AND 850.09  ; 进料伺服X轴#1夹爪配对取放料位标志
AND 851.10  ; 进料伺服Z轴#1夹爪配对取放料位标志
AND W211.01  ; 进料伺服有配对取料需求标志
ORLD
ANDLD
OUT 500.08  ; #1进料夹爪夹紧条件
TIMX(550) 0508 D18  ; 自动运行条件延时时间, #1进料夹爪夹紧延时[A]
LD TR0
LD 500.08  ; #1进料夹爪夹紧条件
AND T0508  ; #1进料夹爪夹紧延时[A]
OR 600.08  ; #1进料夹爪夹紧[A]
ANDLD
ANDNOT 500.09  ; #1进料夹爪松开条件
ANDNOT 300.08  ; #1进料夹爪夹紧[Pls]
ANDNOT 300.09  ; #1进料夹爪松开[Pls]
ANDNOT 800.08  ; #1进料夹爪夹紧位标志[0000.08]
OUT 600.08  ; #1进料夹爪夹紧[A]
LD TR0
LD D1049.03  ; 进料伺服机构#1|2夹爪松开2（步）
AND 850.07  ; 进料伺服X轴#1夹爪扫码NG放料位标志
AND 851.08  ; 进料伺服Z轴#1夹爪扫码NG放料位标志
LD D1052.03  ; 进料伺服机构#1|2夹爪松开|夹紧3（步）
AND 850.09  ; 进料伺服X轴#1夹爪配对取放料位标志
AND 851.10  ; 进料伺服Z轴#1夹爪配对取放料位标志
AND W211.00  ; 进料伺服有配对放料需求标志
ORLD
OR D1055.04  ; 进料伺服机构#1&2夹爪松开4（步）
ANDLD
OUT 500.09  ; #1进料夹爪松开条件
TIMX(550) 0509 D18  ; 自动运行条件延时时间, #1进料夹爪松开延时[A]
LD TR0
LD 500.09  ; #1进料夹爪松开条件
AND T0509  ; #1进料夹爪松开延时[A]
OR 600.09  ; #1进料夹爪松开[A]
ANDLD
ANDNOT 500.08  ; #1进料夹爪夹紧条件
ANDNOT 300.09  ; #1进料夹爪松开[Pls]
ANDNOT 300.08  ; #1进料夹爪夹紧[Pls]
ANDNOT 800.09  ; #1进料夹爪松开位标志[0000.09]
OUT 600.09  ; #1进料夹爪松开[A]

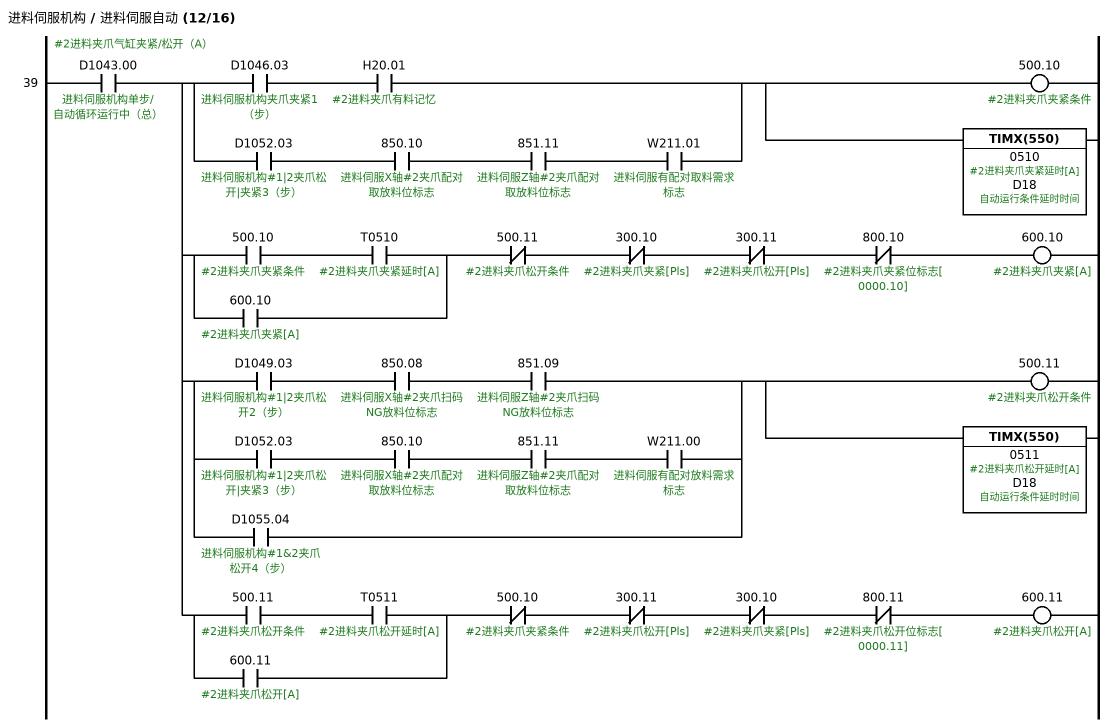
; rung 39: #2进料夹爪气缸夹紧/松开（A）
LD D1043.00  ; 进料伺服机构单步/自动循环运行中（总）
OUT TR0
LD D1046.03  ; 进料伺服机构夹爪夹紧1（步）
AND H20.01  ; #2进料夹爪有料记忆
LD D1052.03  ; 进料伺服机构#1|2夹爪松开|夹紧3（步）
AND 850.10  ; 进料伺服X轴#2夹爪配对取放料位标志
AND 851.11  ; 进料伺服Z轴#2夹爪配对取放料位标志
AND W211.01  ; 进料伺服有配对取料需求标志
ORLD
ANDLD
OUT 500.10  ; #2进料夹爪夹紧条件
TIMX(550) 0510 D18  ; 自动运行条件延时时间, #2进料夹爪夹紧延时[A]
LD TR0
LD 500.10  ; #2进料夹爪夹紧条件
AND T0510  ; #2进料夹爪夹紧延时[A]
OR 600.10  ; #2进料夹爪夹紧[A]
ANDLD
ANDNOT 500.11  ; #2进料夹爪松开条件
ANDNOT 300.10  ; #2进料夹爪夹紧[Pls]
ANDNOT 300.11  ; #2进料夹爪松开[Pls]
ANDNOT 800.10  ; #2进料夹爪夹紧位标志[0000.10]
OUT 600.10  ; #2进料夹爪夹紧[A]
LD TR0
LD D1049.03  ; 进料伺服机构#1|2夹爪松开2（步）
AND 850.08  ; 进料伺服X轴#2夹爪扫码NG放料位标志
AND 851.09  ; 进料伺服Z轴#2夹爪扫码NG放料位标志
LD D1052.03  ; 进料伺服机构#1|2夹爪松开|夹紧3（步）
AND 850.10  ; 进料伺服X轴#2夹爪配对取放料位标志
AND 851.11  ; 进料伺服Z轴#2夹爪配对取放料位标志
AND W211.00  ; 进料伺服有配对放料需求标志
ORLD
OR D1055.04  ; 进料伺服机构#1&2夹爪松开4（步）
ANDLD
OUT 500.11  ; #2进料夹爪松开条件
TIMX(550) 0511 D18  ; 自动运行条件延时时间, #2进料夹爪松开延时[A]
LD TR0
LD 500.11  ; #2进料夹爪松开条件
AND T0511  ; #2进料夹爪松开延时[A]
OR 600.11  ; #2进料夹爪松开[A]
ANDLD
ANDNOT 500.10  ; #2进料夹爪夹紧条件
ANDNOT 300.11  ; #2进料夹爪松开[Pls]
ANDNOT 300.10  ; #2进料夹爪夹紧[Pls]
ANDNOT 800.11  ; #2进料夹爪松开位标志[0000.11]
OUT 600.11  ; #2进料夹爪松开[A]

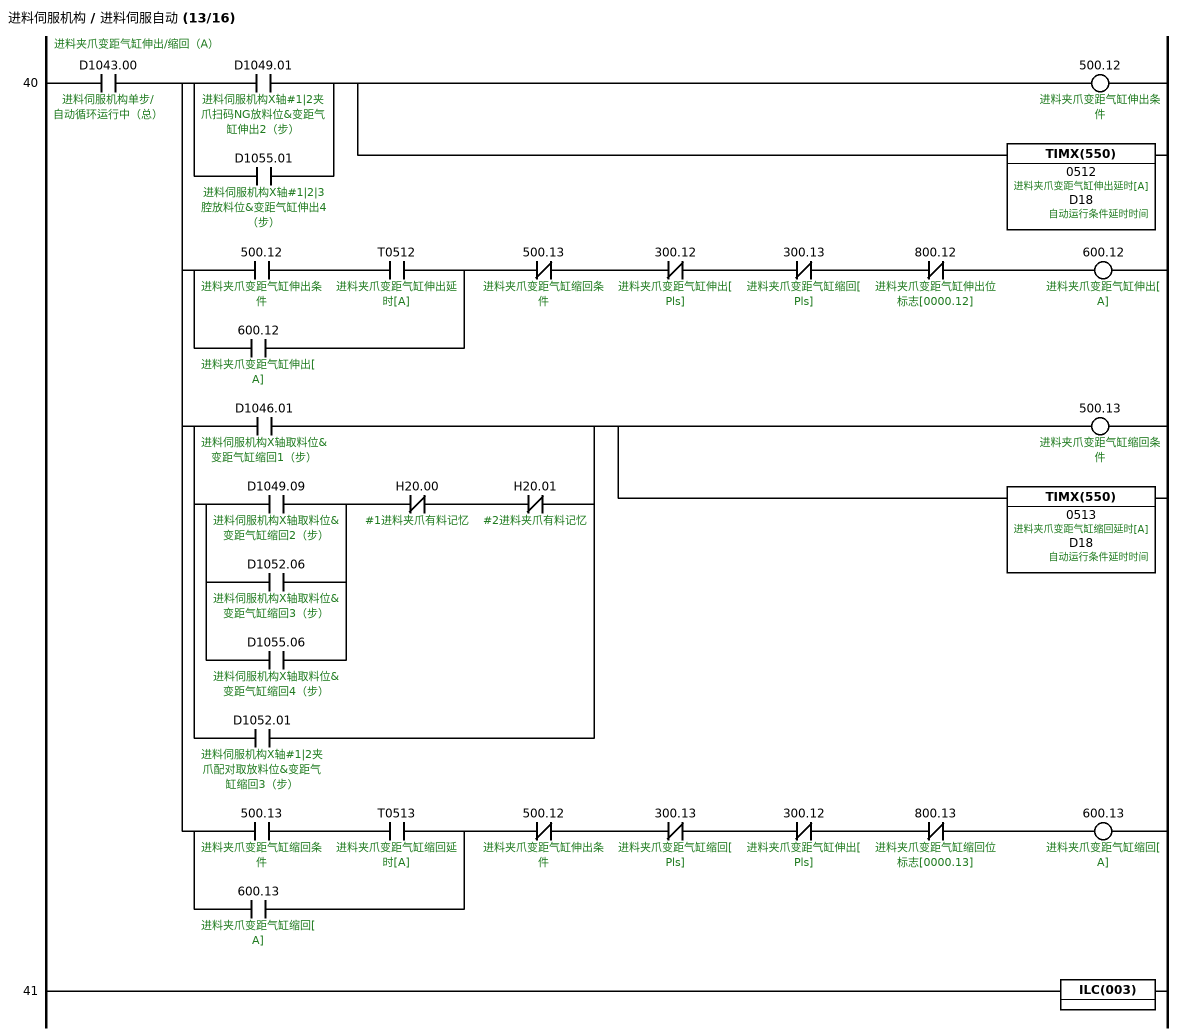
; rung 40: 进料夹爪变距气缸伸出/缩回（A）
LD D1043.00  ; 进料伺服机构单步/自动循环运行中（总）
OUT TR0
LD D1049.01  ; 进料伺服机构X轴#1|2夹爪扫码NG放料位&变距气缸伸出2（步）
OR D1055.01  ; 进料伺服机构X轴#1|2|3腔放料位&变距气缸伸出4（步）
ANDLD
OUT 500.12  ; 进料夹爪变距气缸伸出条件
TIMX(550) 0512 D18  ; 自动运行条件延时时间, 进料夹爪变距气缸伸出延时[A]
LD TR0
LD 500.12  ; 进料夹爪变距气缸伸出条件
AND T0512  ; 进料夹爪变距气缸伸出延时[A]
OR 600.12  ; 进料夹爪变距气缸伸出[A]
ANDLD
ANDNOT 500.13  ; 进料夹爪变距气缸缩回条件
ANDNOT 300.12  ; 进料夹爪变距气缸伸出[Pls]
ANDNOT 300.13  ; 进料夹爪变距气缸缩回[Pls]
ANDNOT 800.12  ; 进料夹爪变距气缸伸出位标志[0000.12]
OUT 600.12  ; 进料夹爪变距气缸伸出[A]
LD TR0
LD D1046.01  ; 进料伺服机构X轴取料位&变距气缸缩回1（步）
LD D1049.09  ; 进料伺服机构X轴取料位&变距气缸缩回2（步）
OR D1052.06  ; 进料伺服机构X轴取料位&变距气缸缩回3（步）
OR D1055.06  ; 进料伺服机构X轴取料位&变距气缸缩回4（步）
ANDNOT H20.00  ; #1进料夹爪有料记忆
ANDNOT H20.01  ; #2进料夹爪有料记忆
ORLD
OR D1052.01  ; 进料伺服机构X轴#1|2夹爪配对取放料位&变距气缸缩回3（步）
ANDLD
OUT 500.13  ; 进料夹爪变距气缸缩回条件
TIMX(550) 0513 D18  ; 自动运行条件延时时间, 进料夹爪变距气缸缩回延时[A]
LD TR0
LD 500.13  ; 进料夹爪变距气缸缩回条件
AND T0513  ; 进料夹爪变距气缸缩回延时[A]
OR 600.13  ; 进料夹爪变距气缸缩回[A]
ANDLD
ANDNOT 500.12  ; 进料夹爪变距气缸伸出条件
ANDNOT 300.13  ; 进料夹爪变距气缸缩回[Pls]
ANDNOT 300.12  ; 进料夹爪变距气缸伸出[Pls]
ANDNOT 800.13  ; 进料夹爪变距气缸缩回位标志[0000.13]
OUT 600.13  ; 进料夹爪变距气缸缩回[A]
; rung 41
ILC(003)

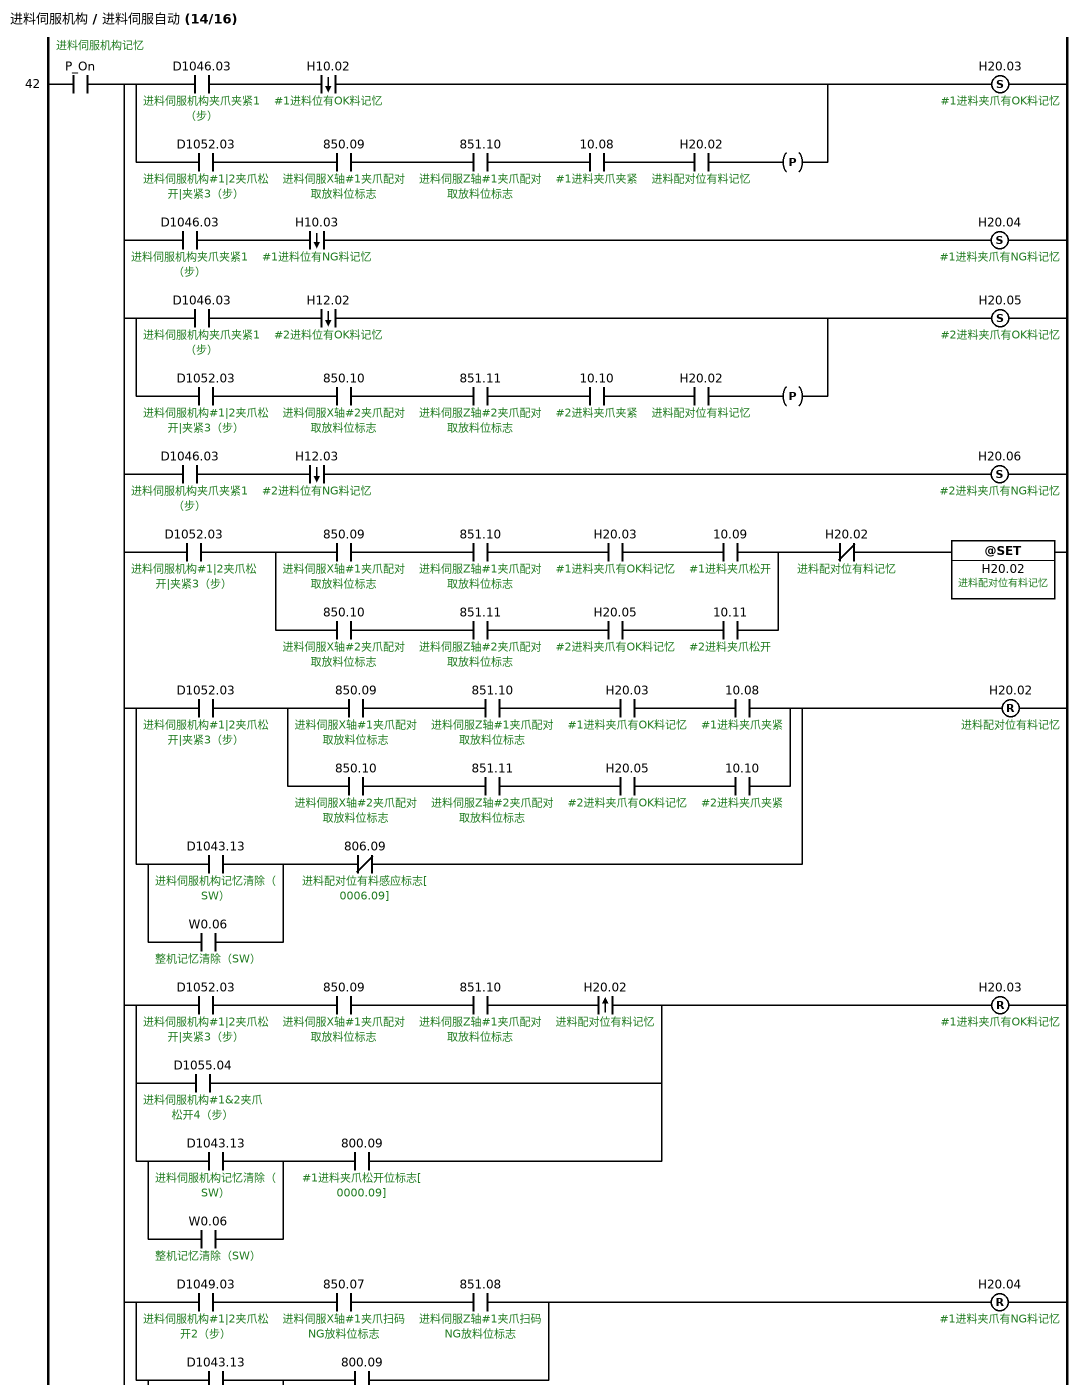

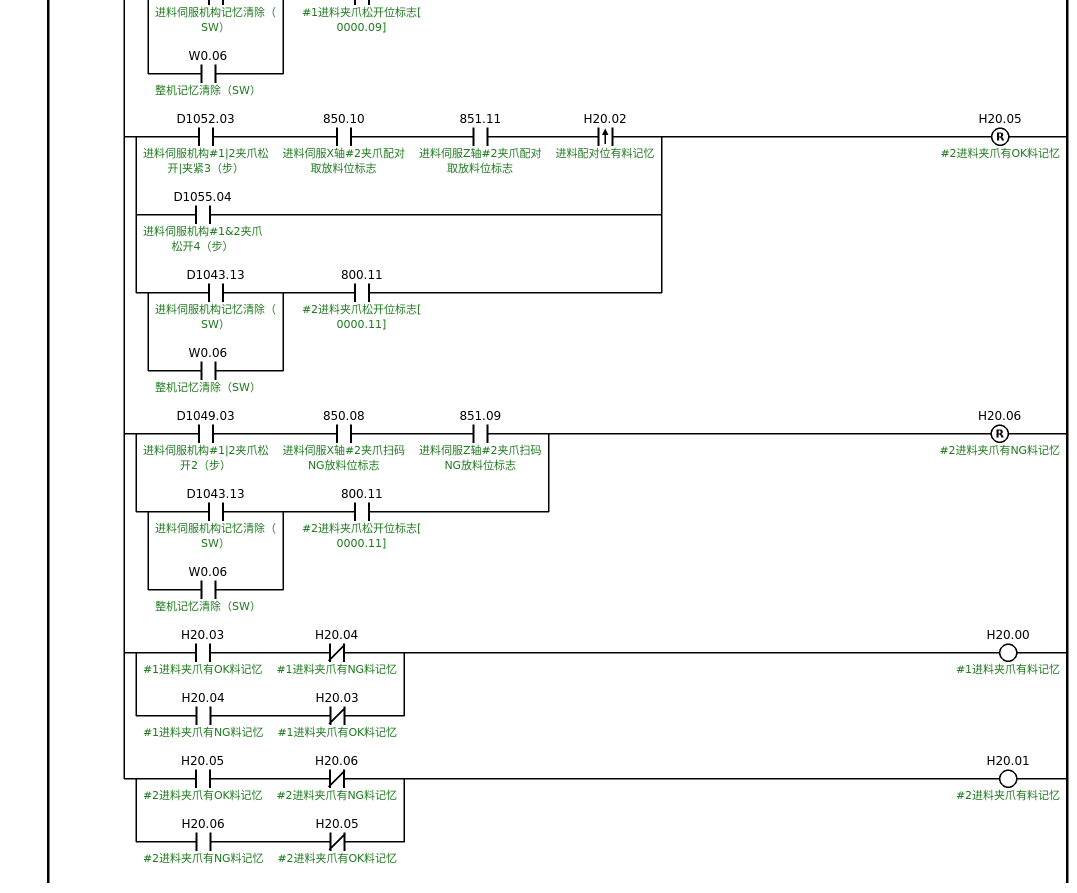
; rung 42: 进料伺服机构记忆
LD P_On
OUT TR0
LD D1046.03  ; 进料伺服机构夹爪夹紧1（步）
%AND H10.02  ; #1进料位有OK料记忆
LD D1052.03  ; 进料伺服机构#1|2夹爪松开|夹紧3（步）
AND 850.09  ; 进料伺服X轴#1夹爪配对取放料位标志
AND 851.10  ; 进料伺服Z轴#1夹爪配对取放料位标志
AND 10.08  ; #1进料夹爪夹紧
AND H20.02  ; 进料配对位有料记忆
UP(521)
ORLD
ANDLD
SET H20.03  ; #1进料夹爪有OK料记忆
LD TR0
AND D1046.03  ; 进料伺服机构夹爪夹紧1（步）
%AND H10.03  ; #1进料位有NG料记忆
SET H20.04  ; #1进料夹爪有NG料记忆
LD TR0
LD D1046.03  ; 进料伺服机构夹爪夹紧1（步）
%AND H12.02  ; #2进料位有OK料记忆
LD D1052.03  ; 进料伺服机构#1|2夹爪松开|夹紧3（步）
AND 850.10  ; 进料伺服X轴#2夹爪配对取放料位标志
AND 851.11  ; 进料伺服Z轴#2夹爪配对取放料位标志
AND 10.10  ; #2进料夹爪夹紧
AND H20.02  ; 进料配对位有料记忆
UP(521)
ORLD
ANDLD
SET H20.05  ; #2进料夹爪有OK料记忆
LD TR0
AND D1046.03  ; 进料伺服机构夹爪夹紧1（步）
%AND H12.03  ; #2进料位有NG料记忆
SET H20.06  ; #2进料夹爪有NG料记忆
LD TR0
AND D1052.03  ; 进料伺服机构#1|2夹爪松开|夹紧3（步）
LD 850.09  ; 进料伺服X轴#1夹爪配对取放料位标志
AND 851.10  ; 进料伺服Z轴#1夹爪配对取放料位标志
AND H20.03  ; #1进料夹爪有OK料记忆
AND 10.09  ; #1进料夹爪松开
LD 850.10  ; 进料伺服X轴#2夹爪配对取放料位标志
AND 851.11  ; 进料伺服Z轴#2夹爪配对取放料位标志
AND H20.05  ; #2进料夹爪有OK料记忆
AND 10.11  ; #2进料夹爪松开
ORLD
ANDLD
ANDNOT H20.02  ; 进料配对位有料记忆
@SET H20.02  ; 进料配对位有料记忆
LD TR0
LD D1052.03  ; 进料伺服机构#1|2夹爪松开|夹紧3（步）
LD 850.09  ; 进料伺服X轴#1夹爪配对取放料位标志
AND 851.10  ; 进料伺服Z轴#1夹爪配对取放料位标志
AND H20.03  ; #1进料夹爪有OK料记忆
AND 10.08  ; #1进料夹爪夹紧
LD 850.10  ; 进料伺服X轴#2夹爪配对取放料位标志
AND 851.11  ; 进料伺服Z轴#2夹爪配对取放料位标志
AND H20.05  ; #2进料夹爪有OK料记忆
AND 10.10  ; #2进料夹爪夹紧
ORLD
ANDLD
LD D1043.13  ; 进料伺服机构记忆清除（SW）
OR W0.06  ; 整机记忆清除（SW）
ANDNOT 806.09  ; 进料配对位有料感应标志[0006.09]
ORLD
ANDLD
RSET H20.02  ; 进料配对位有料记忆
LD TR0
LD D1052.03  ; 进料伺服机构#1|2夹爪松开|夹紧3（步）
AND 850.09  ; 进料伺服X轴#1夹爪配对取放料位标志
AND 851.10  ; 进料伺服Z轴#1夹爪配对取放料位标志
@AND H20.02  ; 进料配对位有料记忆
OR D1055.04  ; 进料伺服机构#1&2夹爪松开4（步）
LD D1043.13  ; 进料伺服机构记忆清除（SW）
OR W0.06  ; 整机记忆清除（SW）
AND 800.09  ; #1进料夹爪松开位标志[0000.09]
ORLD
ANDLD
RSET H20.03  ; #1进料夹爪有OK料记忆
LD TR0
LD D1049.03  ; 进料伺服机构#1|2夹爪松开2（步）
AND 850.07  ; 进料伺服X轴#1夹爪扫码NG放料位标志
AND 851.08  ; 进料伺服Z轴#1夹爪扫码NG放料位标志
LD D1043.13  ; 进料伺服机构记忆清除（SW）
OR W0.06  ; 整机记忆清除（SW）
AND 800.09  ; #1进料夹爪松开位标志[0000.09]
ORLD
ANDLD
RSET H20.04  ; #1进料夹爪有NG料记忆
LD TR0
LD D1052.03  ; 进料伺服机构#1|2夹爪松开|夹紧3（步）
AND 850.10  ; 进料伺服X轴#2夹爪配对取放料位标志
AND 851.11  ; 进料伺服Z轴#2夹爪配对取放料位标志
@AND H20.02  ; 进料配对位有料记忆
OR D1055.04  ; 进料伺服机构#1&2夹爪松开4（步）
LD D1043.13  ; 进料伺服机构记忆清除（SW）
OR W0.06  ; 整机记忆清除（SW）
AND 800.11  ; #2进料夹爪松开位标志[0000.11]
ORLD
ANDLD
RSET H20.05  ; #2进料夹爪有OK料记忆
LD TR0
LD D1049.03  ; 进料伺服机构#1|2夹爪松开2（步）
AND 850.08  ; 进料伺服X轴#2夹爪扫码NG放料位标志
AND 851.09  ; 进料伺服Z轴#2夹爪扫码NG放料位标志
LD D1043.13  ; 进料伺服机构记忆清除（SW）
OR W0.06  ; 整机记忆清除（SW）
AND 800.11  ; #2进料夹爪松开位标志[0000.11]
ORLD
ANDLD
RSET H20.06  ; #2进料夹爪有NG料记忆
LD TR0
LD H20.03  ; #1进料夹爪有OK料记忆
ANDNOT H20.04  ; #1进料夹爪有NG料记忆
LD H20.04  ; #1进料夹爪有NG料记忆
ANDNOT H20.03  ; #1进料夹爪有OK料记忆
ORLD
ANDLD
OUT H20.00  ; #1进料夹爪有料记忆
LD TR0
LD H20.05  ; #2进料夹爪有OK料记忆
ANDNOT H20.06  ; #2进料夹爪有NG料记忆
LD H20.06  ; #2进料夹爪有NG料记忆
ANDNOT H20.05  ; #2进料夹爪有OK料记忆
ORLD
ANDLD
OUT H20.01  ; #2进料夹爪有料记忆

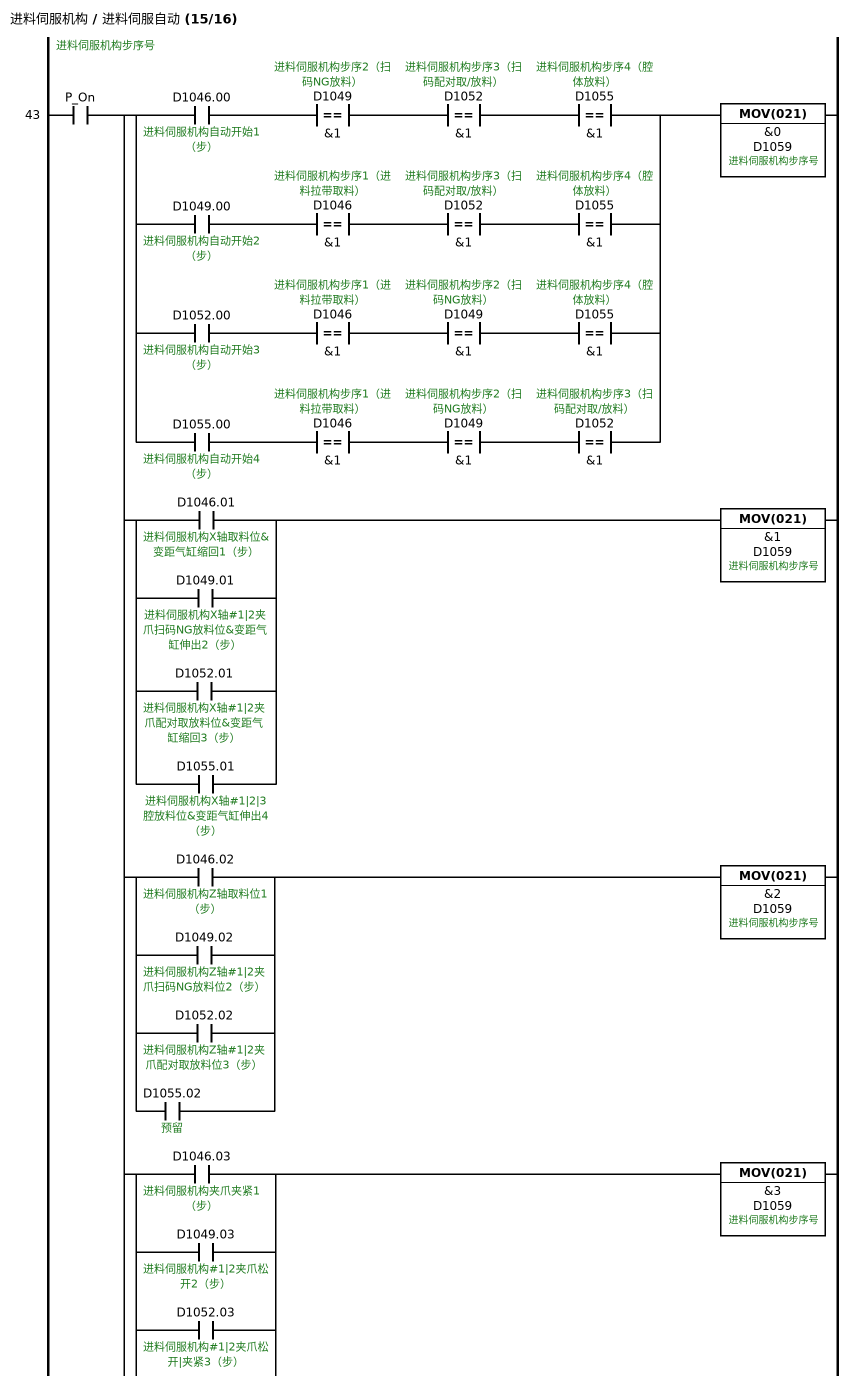

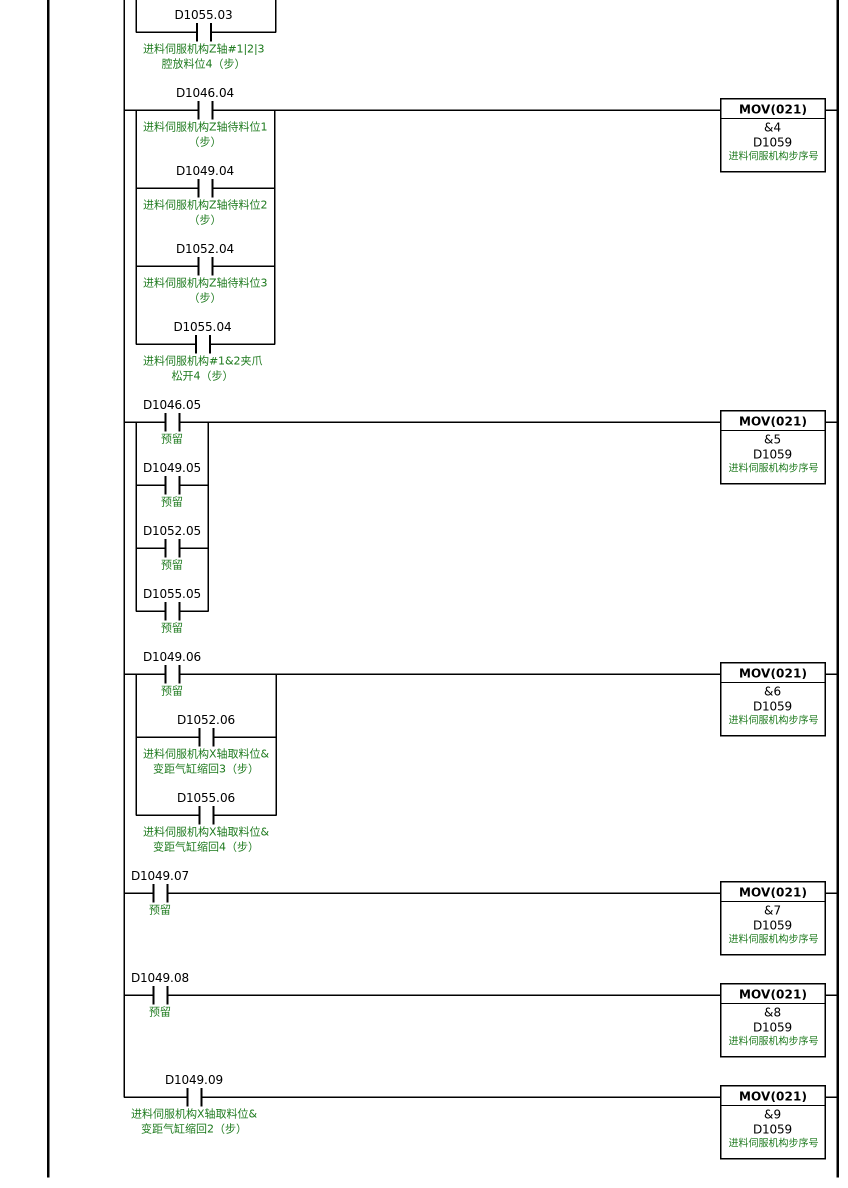
; rung 43: 进料伺服机构步序号
LD P_On
OUT TR0
LD D1046.00  ; 进料伺服机构自动开始1（步）
AND=(300) D1049 &1  ; 进料伺服机构步序2（扫码NG放料）
AND=(300) D1052 &1  ; 进料伺服机构步序3（扫码配对取/放料）
AND=(300) D1055 &1  ; 进料伺服机构步序4（腔体放料）
LD D1049.00  ; 进料伺服机构自动开始2（步）
AND=(300) D1046 &1  ; 进料伺服机构步序1（进料拉带取料）
AND=(300) D1052 &1  ; 进料伺服机构步序3（扫码配对取/放料）
AND=(300) D1055 &1  ; 进料伺服机构步序4（腔体放料）
ORLD
LD D1052.00  ; 进料伺服机构自动开始3（步）
AND=(300) D1046 &1  ; 进料伺服机构步序1（进料拉带取料）
AND=(300) D1049 &1  ; 进料伺服机构步序2（扫码NG放料）
AND=(300) D1055 &1  ; 进料伺服机构步序4（腔体放料）
ORLD
LD D1055.00  ; 进料伺服机构自动开始4（步）
AND=(300) D1046 &1  ; 进料伺服机构步序1（进料拉带取料）
AND=(300) D1049 &1  ; 进料伺服机构步序2（扫码NG放料）
AND=(300) D1052 &1  ; 进料伺服机构步序3（扫码配对取/放料）
ORLD
ANDLD
MOV(021) &0 D1059  ; 进料伺服机构步序号
LD TR0
LD D1046.01  ; 进料伺服机构X轴取料位&变距气缸缩回1（步）
OR D1049.01  ; 进料伺服机构X轴#1|2夹爪扫码NG放料位&变距气缸伸出2（步）
OR D1052.01  ; 进料伺服机构X轴#1|2夹爪配对取放料位&变距气缸缩回3（步）
OR D1055.01  ; 进料伺服机构X轴#1|2|3腔放料位&变距气缸伸出4（步）
ANDLD
MOV(021) &1 D1059  ; 进料伺服机构步序号
LD TR0
LD D1046.02  ; 进料伺服机构Z轴取料位1（步）
OR D1049.02  ; 进料伺服机构Z轴#1|2夹爪扫码NG放料位2（步）
OR D1052.02  ; 进料伺服机构Z轴#1|2夹爪配对取放料位3（步）
OR D1055.02  ; 预留
ANDLD
MOV(021) &2 D1059  ; 进料伺服机构步序号
LD TR0
LD D1046.03  ; 进料伺服机构夹爪夹紧1（步）
OR D1049.03  ; 进料伺服机构#1|2夹爪松开2（步）
OR D1052.03  ; 进料伺服机构#1|2夹爪松开|夹紧3（步）
OR D1055.03  ; 进料伺服机构Z轴#1|2|3腔放料位4（步）
ANDLD
MOV(021) &3 D1059  ; 进料伺服机构步序号
LD TR0
LD D1046.04  ; 进料伺服机构Z轴待料位1（步）
OR D1049.04  ; 进料伺服机构Z轴待料位2（步）
OR D1052.04  ; 进料伺服机构Z轴待料位3（步）
OR D1055.04  ; 进料伺服机构#1&2夹爪松开4（步）
ANDLD
MOV(021) &4 D1059  ; 进料伺服机构步序号
LD TR0
LD D1046.05  ; 预留
OR D1049.05  ; 预留
OR D1052.05  ; 预留
OR D1055.05  ; 预留
ANDLD
MOV(021) &5 D1059  ; 进料伺服机构步序号
LD TR0
LD D1049.06  ; 预留
OR D1052.06  ; 进料伺服机构X轴取料位&变距气缸缩回3（步）
OR D1055.06  ; 进料伺服机构X轴取料位&变距气缸缩回4（步）
ANDLD
MOV(021) &6 D1059  ; 进料伺服机构步序号
LD TR0
AND D1049.07  ; 预留
MOV(021) &7 D1059  ; 进料伺服机构步序号
LD TR0
AND D1049.08  ; 预留
MOV(021) &8 D1059  ; 进料伺服机构步序号
LD TR0
AND D1049.09  ; 进料伺服机构X轴取料位&变距气缸缩回2（步）
MOV(021) &9 D1059  ; 进料伺服机构步序号

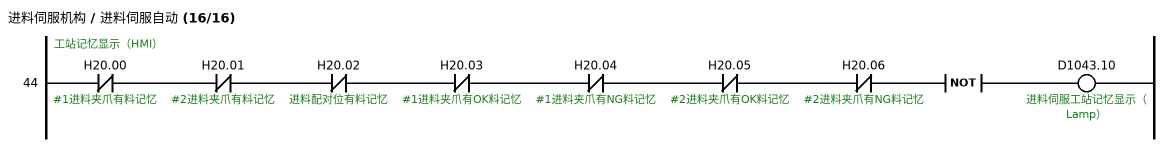
; rung 44: 工站记忆显示（HMI）
LDNOT H20.00  ; #1进料夹爪有料记忆
ANDNOT H20.01  ; #2进料夹爪有料记忆
ANDNOT H20.02  ; 进料配对位有料记忆
ANDNOT H20.03  ; #1进料夹爪有OK料记忆
ANDNOT H20.04  ; #1进料夹爪有NG料记忆
ANDNOT H20.05  ; #2进料夹爪有OK料记忆
ANDNOT H20.06  ; #2进料夹爪有NG料记忆
NOT(520)
OUT D1043.10  ; 进料伺服工站记忆显示（Lamp）

### Section 工站复位

